(*-------------------------------------------------------------------------------------------------------ЕСЛИ ВТОРАЯ ГОРЕЛКА 1*)
	IF SECOND_GORELKA=1 THEN
		 IF AVARIA_OSNOVNAYA_GORELKA=FALSE  AND AVARIA_SECOND_GORELKA=FALSE THEN
			IF TEMPERATURA_2_OBR_OTOPLENIYA_AI_SP_307<TEMPERATURA_OFF_CIRCULACIONNOGO_NASOSA THEN
				xDO8:=TRUE;
				STEP_CIRCULAYCIONNUY_NASOS_1:=1;
			ELSE
				xDO8:=FALSE;
			END_IF
		END_IF
	END_IF
(*--------------------------------------------------------------------ЕСЛИ ВТОРАЯ ГОРЕЛКА 1 И ОСНОВНАЯ ВЫШЛА ИЗ СТРОЯ*)
	IF SECOND_GORELKA=1 THEN
		 IF AVARIA_OSNOVNAYA_GORELKA=TRUE  AND AVARIA_SECOND_GORELKA=FALSE THEN
			xDO8:=TRUE;
			STEP_CIRCULAYCIONNUY_NASOS_1:=1;
		END_IF
	END_IF
(*--------------------------------------------------------------------ЕСЛИ РЕЗЕРВНАЯ ГОРЕЛКА 1 И ВТОРАЯ ВЫШЛА ИЗ СТРОЯ*)
	IF RESERV_GORELKA=1 THEN
		 IF AVARIA_OSNOVNAYA_GORELKA=TRUE AND AVARIA_SECOND_GORELKA=TRUE THEN
			xDO8:=TRUE;
			STEP_CIRCULAYCIONNUY_NASOS_1:=1;
		END_IF
	END_IF
(*-------------------------------------------------------------------------------------------------------ЕСЛИ РЕЗЕРВНАЯ ГОРЕЛКА 1*)
	IF RESERV_GORELKA=1 THEN
		 IF TEMPERATURA_2_OBR_OTOPLENIYA_AI_SP_307<TEMPERATURA_OFF_CIRCULACIONNOGO_NASOSA THEN
				xDO8:=TRUE;
				STEP_CIRCULAYCIONNUY_NASOS_1:=1;
			ELSE
				xDO8:=FALSE;
			END_IF
	END_IF
END_IF
(*---------------------------------------------------------------------------------РАБОТА НАСОСОСА ПОСЛЕ ОСТАНОВКИ КОТЛА*)
IF PUSK_GORELKA_1=FALSE AND STEP_CIRCULAYCIONNUY_NASOS_1=1 THEN
	CASE STEP_CIRCULAYCIONNUY_NASOS_1 OF
		1:
			TIMER_CIRCUL_NASOS_1(IN:=TRUE,PT:=REAL_TO_TIME(VREMYA_RABOTU_CIRCULYACIONNOGO_NASOSA*1000));
				IF  TIMER_CIRCUL_NASOS_1.ET=TIMER_CIRCUL_NASOS_1.PT THEN
					STEP_CIRCULAYCIONNUY_NASOS_1:=0;
					TIMER_CIRCUL_NASOS_1(IN:=FALSE,PT:=T#0s);
      		 			TIMER_CIRCUL_NASOS_1;
					xDO8:=FALSE;
				END_IF
	END_CASE
ELSE
	TIMER_CIRCUL_NASOS_1(IN:=FALSE,PT:=T#0s);
      	TIMER_CIRCUL_NASOS_1;
END_IF
END_ACTION
ACTION CIRKULYACIONIY_NASOS_2:
IF PUSK_GORELKA_2=TRUE  THEN
(*---------------------------------------------------------------------------------------------------ЕСЛИ ОСНОВНАЯ ГОРЕЛКА 1*)
	IF  OSNOVNAYA_GORELKA=2  THEN
		xDO9:=TRUE;
		STEP_CIRCULAYCIONNUY_NASOS_2:=1;
	END_IF

(*-------------------------------------------------------------------------------------------------------ЕСЛИ ВТОРАЯ ГОРЕЛКА 1*)
	IF SECOND_GORELKA=2 THEN
		 IF AVARIA_OSNOVNAYA_GORELKA=FALSE  AND AVARIA_SECOND_GORELKA=FALSE THEN
			IF TEMPERATURA_2_OBR_OTOPLENIYA_AI_SP_307<TEMPERATURA_OFF_CIRCULACIONNOGO_NASOSA THEN
				xDO9:=TRUE;
				STEP_CIRCULAYCIONNUY_NASOS_2:=1;
			ELSE
				xDO9:=FALSE;
			END_IF
		END_IF
	END_IF
(*--------------------------------------------------------------------ЕСЛИ ВТОРАЯ ГОРЕЛКА 1 И ОСНОВНАЯ ВЫШЛА ИЗ СТРОЯ*)
	IF SECOND_GORELKA=2 THEN
		 IF AVARIA_OSNOVNAYA_GORELKA=TRUE  AND AVARIA_SECOND_GORELKA=FALSE THEN
			xDO9:=TRUE;
			STEP_CIRCULAYCIONNUY_NASOS_2:=1;
		END_IF
	END_IF
(*--------------------------------------------------------------------ЕСЛИ РЕЗЕРВНАЯ ГОРЕЛКА 1 И ВТОРАЯ ВЫШЛА ИЗ СТРОЯ*)
	IF RESERV_GORELKA=2 THEN
		 IF AVARIA_OSNOVNAYA_GORELKA=TRUE AND AVARIA_SECOND_GORELKA=TRUE THEN
			xDO9:=TRUE;
			STEP_CIRCULAYCIONNUY_NASOS_2:=1;
		END_IF
	END_IF
(*-------------------------------------------------------------------------------------------------------ЕСЛИ РЕЗЕРВНАЯ ГОРЕЛКА 1*)
	IF RESERV_GORELKA=2 THEN
		 IF TEMPERATURA_2_OBR_OTOPLENIYA_AI_SP_307<TEMPERATURA_OFF_CIRCULACIONNOGO_NASOSA THEN
				xDO9:=TRUE;
				STEP_CIRCULAYCIONNUY_NASOS_2:=1;
			ELSE
				xDO9:=FALSE;
			END_IF
	END_IF
END_IF
(*---------------------------------------------------------------------------------РАБОТА НАСОСОСА ПОСЛЕ ОСТАНОВКИ КОТЛА*)
IF PUSK_GORELKA_2=FALSE AND STEP_CIRCULAYCIONNUY_NASOS_2=1 THEN
	CASE STEP_CIRCULAYCIONNUY_NASOS_2 OF
		1:
			TIMER_CIRCUL_NASOS_2(IN:=TRUE,PT:=REAL_TO_TIME(VREMYA_RABOTU_CIRCULYACIONNOGO_NASOSA*1000));
				IF  TIMER_CIRCUL_NASOS_2.ET=TIMER_CIRCUL_NASOS_2.PT THEN
					STEP_CIRCULAYCIONNUY_NASOS_2:=0;
					TIMER_CIRCUL_NASOS_2(IN:=FALSE,PT:=T#0s);
      		 			TIMER_CIRCUL_NASOS_2;
					xDO9:=FALSE;
				END_IF
	END_CASE
ELSE
	TIMER_CIRCUL_NASOS_2(IN:=FALSE,PT:=T#0s);
      	TIMER_CIRCUL_NASOS_2;
END_IF
END_ACTION
ACTION CIRKULYACIONIY_NASOS_3:
IF PUSK_GORELKA_3=TRUE  THEN
(*---------------------------------------------------------------------------------------------------ЕСЛИ ОСНОВНАЯ ГОРЕЛКА 1*)
	IF  OSNOVNAYA_GORELKA=3  THEN
		xDO10:=TRUE;
		STEP_CIRCULAYCIONNUY_NASOS_3:=1;
	END_IF

(*-------------------------------------------------------------------------------------------------------ЕСЛИ ВТОРАЯ ГОРЕЛКА 1*)
	IF SECOND_GORELKA=3 THEN
		 IF AVARIA_OSNOVNAYA_GORELKA=FALSE  AND AVARIA_SECOND_GORELKA=FALSE THEN
			IF TEMPERATURA_2_OBR_OTOPLENIYA_AI_SP_307<TEMPERATURA_OFF_CIRCULACIONNOGO_NASOSA THEN
				xDO10:=TRUE;
				STEP_CIRCULAYCIONNUY_NASOS_3:=1;
			ELSE
				xDO10:=FALSE;
			END_IF
		END_IF
	END_IF
(*--------------------------------------------------------------------ЕСЛИ ВТОРАЯ ГОРЕЛКА 1 И ОСНОВНАЯ ВЫШЛА ИЗ СТРОЯ*)
	IF SECOND_GORELKA=3 THEN
		 IF AVARIA_OSNOVNAYA_GORELKA=TRUE  AND AVARIA_SECOND_GORELKA=FALSE THEN
			xDO10:=TRUE;
			STEP_CIRCULAYCIONNUY_NASOS_3:=1;
		END_IF
	END_IF
(*--------------------------------------------------------------------ЕСЛИ РЕЗЕРВНАЯ ГОРЕЛКА 1 И ВТОРАЯ ВЫШЛА ИЗ СТРОЯ*)
	IF RESERV_GORELKA=3 THEN
		 IF AVARIA_OSNOVNAYA_GORELKA=TRUE AND AVARIA_SECOND_GORELKA=TRUE THEN
			xDO10:=TRUE;
			STEP_CIRCULAYCIONNUY_NASOS_3:=1;
		END_IF
	END_IF
(*-------------------------------------------------------------------------------------------------------ЕСЛИ РЕЗЕРВНАЯ ГОРЕЛКА 1*)
	IF RESERV_GORELKA=3 THEN
		 IF TEMPERATURA_2_OBR_OTOPLENIYA_AI_SP_307<TEMPERATURA_OFF_CIRCULACIONNOGO_NASOSA THEN
				xDO10:=TRUE;
				STEP_CIRCULAYCIONNUY_NASOS_3:=1;
			ELSE
				xDO10:=FALSE;
			END_IF
	END_IF
END_IF
(*---------------------------------------------------------------------------------РАБОТА НАСОСОСА ПОСЛЕ ОСТАНОВКИ КОТЛА*)
IF PUSK_GORELKA_3=FALSE AND STEP_CIRCULAYCIONNUY_NASOS_3=1 THEN
	CASE STEP_CIRCULAYCIONNUY_NASOS_3 OF
		1:
			TIMER_CIRCUL_NASOS_3(IN:=TRUE,PT:=REAL_TO_TIME(VREMYA_RABOTU_CIRCULYACIONNOGO_NASOSA*1000));
				IF  TIMER_CIRCUL_NASOS_3.ET=TIMER_CIRCUL_NASOS_3.PT THEN
					STEP_CIRCULAYCIONNUY_NASOS_3:=0;
					TIMER_CIRCUL_NASOS_3(IN:=FALSE,PT:=T#0s);
      		 			TIMER_CIRCUL_NASOS_3;
					xDO10:=FALSE;
				END_IF
	END_CASE
ELSE
	TIMER_CIRCUL_NASOS_3(IN:=FALSE,PT:=T#0s);
      	TIMER_CIRCUL_NASOS_3;
END_IF
END_ACTION
ACTION DECOD_ERROR:
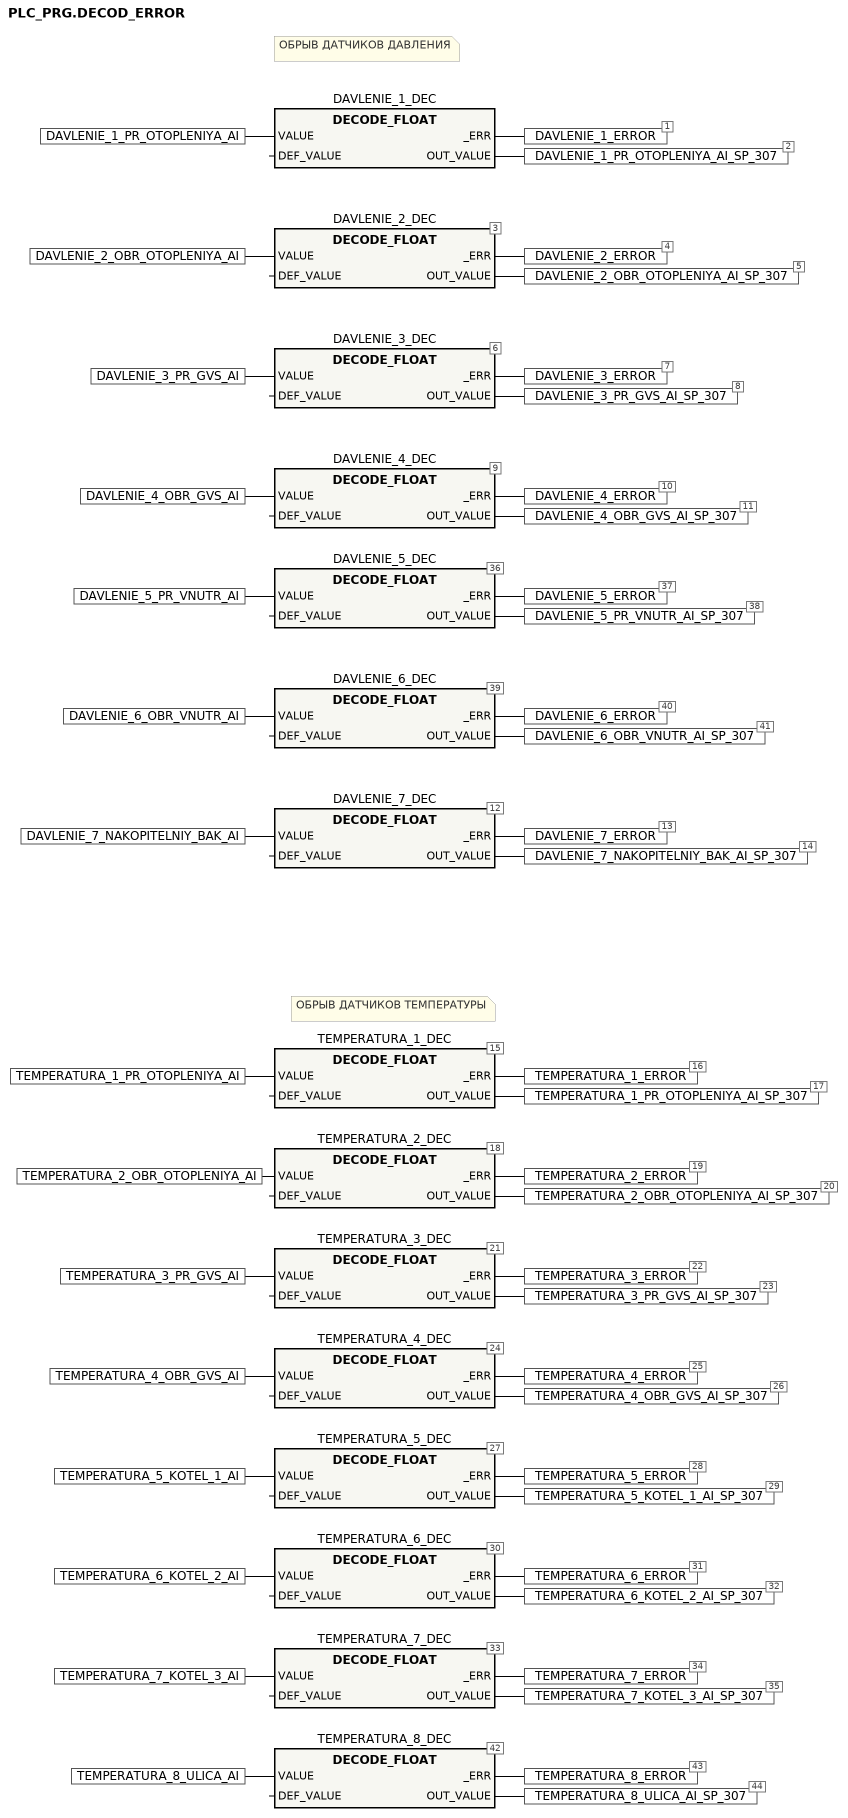
[picture p1: PLC_PRG.DECOD_ERROR (CFC)]
_CFC_ (* Continuous Function Chart, elements in execution order *)
(* ОБРЫВ ДАТЧИКОВ ДАВЛЕНИЯ *)
#0 DAVLENIE_1_DEC:DECODE_FLOAT(VALUE: DAVLENIE_1_PR_OTOPLENIYA_AI, DEF_VALUE: -)
#1 DAVLENIE_1_ERROR <= #0._ERR
#2 DAVLENIE_1_PR_OTOPLENIYA_AI_SP_307 <= #0.OUT_VALUE
#3 DAVLENIE_2_DEC:DECODE_FLOAT(VALUE: DAVLENIE_2_OBR_OTOPLENIYA_AI, DEF_VALUE: -)
#4 DAVLENIE_2_ERROR <= #3._ERR
#5 DAVLENIE_2_OBR_OTOPLENIYA_AI_SP_307 <= #3.OUT_VALUE
#6 DAVLENIE_3_DEC:DECODE_FLOAT(VALUE: DAVLENIE_3_PR_GVS_AI, DEF_VALUE: -)
#7 DAVLENIE_3_ERROR <= #6._ERR
#8 DAVLENIE_3_PR_GVS_AI_SP_307 <= #6.OUT_VALUE
#9 DAVLENIE_4_DEC:DECODE_FLOAT(VALUE: DAVLENIE_4_OBR_GVS_AI, DEF_VALUE: -)
#10 DAVLENIE_4_ERROR <= #9._ERR
#11 DAVLENIE_4_OBR_GVS_AI_SP_307 <= #9.OUT_VALUE
#12 DAVLENIE_7_DEC:DECODE_FLOAT(VALUE: DAVLENIE_7_NAKOPITELNIY_BAK_AI, DEF_VALUE: -)
#13 DAVLENIE_7_ERROR <= #12._ERR
#14 DAVLENIE_7_NAKOPITELNIY_BAK_AI_SP_307 <= #12.OUT_VALUE
#15 TEMPERATURA_1_DEC:DECODE_FLOAT(VALUE: TEMPERATURA_1_PR_OTOPLENIYA_AI, DEF_VALUE: -)
#16 TEMPERATURA_1_ERROR <= #15._ERR
#17 TEMPERATURA_1_PR_OTOPLENIYA_AI_SP_307 <= #15.OUT_VALUE
#18 TEMPERATURA_2_DEC:DECODE_FLOAT(VALUE: TEMPERATURA_2_OBR_OTOPLENIYA_AI, DEF_VALUE: -)
#19 TEMPERATURA_2_ERROR <= #18._ERR
#20 TEMPERATURA_2_OBR_OTOPLENIYA_AI_SP_307 <= #18.OUT_VALUE
#21 TEMPERATURA_3_DEC:DECODE_FLOAT(VALUE: TEMPERATURA_3_PR_GVS_AI, DEF_VALUE: -)
#22 TEMPERATURA_3_ERROR <= #21._ERR
#23 TEMPERATURA_3_PR_GVS_AI_SP_307 <= #21.OUT_VALUE
#24 TEMPERATURA_4_DEC:DECODE_FLOAT(VALUE: TEMPERATURA_4_OBR_GVS_AI, DEF_VALUE: -)
#25 TEMPERATURA_4_ERROR <= #24._ERR
#26 TEMPERATURA_4_OBR_GVS_AI_SP_307 <= #24.OUT_VALUE
#27 TEMPERATURA_5_DEC:DECODE_FLOAT(VALUE: TEMPERATURA_5_KOTEL_1_AI, DEF_VALUE: -)
#28 TEMPERATURA_5_ERROR <= #27._ERR
#29 TEMPERATURA_5_KOTEL_1_AI_SP_307 <= #27.OUT_VALUE
#30 TEMPERATURA_6_DEC:DECODE_FLOAT(VALUE: TEMPERATURA_6_KOTEL_2_AI, DEF_VALUE: -)
#31 TEMPERATURA_6_ERROR <= #30._ERR
#32 TEMPERATURA_6_KOTEL_2_AI_SP_307 <= #30.OUT_VALUE
#33 TEMPERATURA_7_DEC:DECODE_FLOAT(VALUE: TEMPERATURA_7_KOTEL_3_AI, DEF_VALUE: -)
#34 TEMPERATURA_7_ERROR <= #33._ERR
#35 TEMPERATURA_7_KOTEL_3_AI_SP_307 <= #33.OUT_VALUE
(* ОБРЫВ ДАТЧИКОВ ТЕМПЕРАТУРЫ *)
#36 DAVLENIE_5_DEC:DECODE_FLOAT(VALUE: DAVLENIE_5_PR_VNUTR_AI, DEF_VALUE: -)
#37 DAVLENIE_5_ERROR <= #36._ERR
#38 DAVLENIE_5_PR_VNUTR_AI_SP_307 <= #36.OUT_VALUE
#39 DAVLENIE_6_DEC:DECODE_FLOAT(VALUE: DAVLENIE_6_OBR_VNUTR_AI, DEF_VALUE: -)
#40 DAVLENIE_6_ERROR <= #39._ERR
#41 DAVLENIE_6_OBR_VNUTR_AI_SP_307 <= #39.OUT_VALUE
#42 TEMPERATURA_8_DEC:DECODE_FLOAT(VALUE: TEMPERATURA_8_ULICA_AI, DEF_VALUE: -)
#43 TEMPERATURA_8_ERROR <= #42._ERR
#44 TEMPERATURA_8_ULICA_AI_SP_307 <= #42.OUT_VALUE
_END_CFC_
(* the same logic as Structured Text *)
(* ОБРЫВ ДАТЧИКОВ ДАВЛЕНИЯ *)
DAVLENIE_1_DEC(VALUE := DAVLENIE_1_PR_OTOPLENIYA_AI);
DAVLENIE_1_ERROR := DAVLENIE_1_DEC._ERR;
DAVLENIE_1_PR_OTOPLENIYA_AI_SP_307 := DAVLENIE_1_DEC.OUT_VALUE;
DAVLENIE_2_DEC(VALUE := DAVLENIE_2_OBR_OTOPLENIYA_AI);
DAVLENIE_2_ERROR := DAVLENIE_2_DEC._ERR;
DAVLENIE_2_OBR_OTOPLENIYA_AI_SP_307 := DAVLENIE_2_DEC.OUT_VALUE;
DAVLENIE_3_DEC(VALUE := DAVLENIE_3_PR_GVS_AI);
DAVLENIE_3_ERROR := DAVLENIE_3_DEC._ERR;
DAVLENIE_3_PR_GVS_AI_SP_307 := DAVLENIE_3_DEC.OUT_VALUE;
DAVLENIE_4_DEC(VALUE := DAVLENIE_4_OBR_GVS_AI);
DAVLENIE_4_ERROR := DAVLENIE_4_DEC._ERR;
DAVLENIE_4_OBR_GVS_AI_SP_307 := DAVLENIE_4_DEC.OUT_VALUE;
DAVLENIE_7_DEC(VALUE := DAVLENIE_7_NAKOPITELNIY_BAK_AI);
DAVLENIE_7_ERROR := DAVLENIE_7_DEC._ERR;
DAVLENIE_7_NAKOPITELNIY_BAK_AI_SP_307 := DAVLENIE_7_DEC.OUT_VALUE;
TEMPERATURA_1_DEC(VALUE := TEMPERATURA_1_PR_OTOPLENIYA_AI);
TEMPERATURA_1_ERROR := TEMPERATURA_1_DEC._ERR;
TEMPERATURA_1_PR_OTOPLENIYA_AI_SP_307 := TEMPERATURA_1_DEC.OUT_VALUE;
TEMPERATURA_2_DEC(VALUE := TEMPERATURA_2_OBR_OTOPLENIYA_AI);
TEMPERATURA_2_ERROR := TEMPERATURA_2_DEC._ERR;
TEMPERATURA_2_OBR_OTOPLENIYA_AI_SP_307 := TEMPERATURA_2_DEC.OUT_VALUE;
TEMPERATURA_3_DEC(VALUE := TEMPERATURA_3_PR_GVS_AI);
TEMPERATURA_3_ERROR := TEMPERATURA_3_DEC._ERR;
TEMPERATURA_3_PR_GVS_AI_SP_307 := TEMPERATURA_3_DEC.OUT_VALUE;
TEMPERATURA_4_DEC(VALUE := TEMPERATURA_4_OBR_GVS_AI);
TEMPERATURA_4_ERROR := TEMPERATURA_4_DEC._ERR;
TEMPERATURA_4_OBR_GVS_AI_SP_307 := TEMPERATURA_4_DEC.OUT_VALUE;
TEMPERATURA_5_DEC(VALUE := TEMPERATURA_5_KOTEL_1_AI);
TEMPERATURA_5_ERROR := TEMPERATURA_5_DEC._ERR;
TEMPERATURA_5_KOTEL_1_AI_SP_307 := TEMPERATURA_5_DEC.OUT_VALUE;
TEMPERATURA_6_DEC(VALUE := TEMPERATURA_6_KOTEL_2_AI);
TEMPERATURA_6_ERROR := TEMPERATURA_6_DEC._ERR;
TEMPERATURA_6_KOTEL_2_AI_SP_307 := TEMPERATURA_6_DEC.OUT_VALUE;
TEMPERATURA_7_DEC(VALUE := TEMPERATURA_7_KOTEL_3_AI);
TEMPERATURA_7_ERROR := TEMPERATURA_7_DEC._ERR;
TEMPERATURA_7_KOTEL_3_AI_SP_307 := TEMPERATURA_7_DEC.OUT_VALUE;
(* ОБРЫВ ДАТЧИКОВ ТЕМПЕРАТУРЫ *)
DAVLENIE_5_DEC(VALUE := DAVLENIE_5_PR_VNUTR_AI);
DAVLENIE_5_ERROR := DAVLENIE_5_DEC._ERR;
DAVLENIE_5_PR_VNUTR_AI_SP_307 := DAVLENIE_5_DEC.OUT_VALUE;
DAVLENIE_6_DEC(VALUE := DAVLENIE_6_OBR_VNUTR_AI);
DAVLENIE_6_ERROR := DAVLENIE_6_DEC._ERR;
DAVLENIE_6_OBR_VNUTR_AI_SP_307 := DAVLENIE_6_DEC.OUT_VALUE;
TEMPERATURA_8_DEC(VALUE := TEMPERATURA_8_ULICA_AI);
TEMPERATURA_8_ERROR := TEMPERATURA_8_DEC._ERR;
TEMPERATURA_8_ULICA_AI_SP_307 := TEMPERATURA_8_DEC.OUT_VALUE;
END_ACTION
ACTION DO_DISKRETNUY_OUT:
xDO.0:=xDO0;
xDO.1:=xDO1;
xDO.2:=xDO2;
xDO.3:=xDO3;
xDO.4:=xDO4;
xDO.5:=xDO5;
xDO.6:=xDO6;
xDO.7:=xDO7;
xDO.8:=xDO8;
xDO.9:=xDO9;
xDO.10:=xDO10;
xDO.11:=xDO11;
xDO.12:=xDO12;
xDO.13:=xDO13;
xDO.14:=xDO14;
xDO.15:=xDO15;
END_ACTION
ACTION KASKAD_GORELOK:
UPRAVLENIE_GORELKOY_1;
UPRAVLENIE_GORELKOY_2;
UPRAVLENIE_GORELKOY_3;

IF WORK_KASKAD_1_SETEVOY=FALSE THEN
	PUSK_GORELKA_1:=FALSE;
	PUSK_GORELKA_2:=FALSE;
	PUSK_GORELKA_3:=FALSE;
END_IF
END_ACTION
ACTION MODUL_ERROR:
(*CASE STEP_MODUL_ERROR OF
0:
	IF ERROR_CONNECT<>0 THEN
		STEP_MODUL_ERROR:=1;
	END_IF
1:
	TIMER_MODUL_ERROR(IN:=TRUE, PT:=T#5s);
			IF  TIMER_MODUL_ERROR.ET=TIMER_MODUL_ERROR.PT THEN
				IF ERROR_CONNECT<>0 THEN
						ERROR_MODUL_SP_307:=TRUE;
						STEP_MODUL_ERROR:=0;
						TIMER_MODUL_ERROR(IN:=FALSE,PT:=T#0s);
      						TIMER_MODUL_ERROR;
				ELSE
					ERROR_MODUL_SP_307:=FALSE;
					STEP_MODUL_ERROR:=0;
					TIMER_MODUL_ERROR(IN:=FALSE,PT:=T#0s);
      					TIMER_MODUL_ERROR;
				END_IF
				TIMER_MODUL_ERROR(IN:=FALSE,PT:=T#0s);
      		 		TIMER_MODUL_ERROR;
			END_IF
END_CASE
*)

CASE STEP_MODUL_ERROR OF
0:
	IF ERROR_CONNECT<>0 THEN
		STEP_MODUL_ERROR:=1;
	END_IF
1:
	TIMER_MODUL_ERROR(IN:=TRUE, PT:=T#15s);
		IF  TIMER_MODUL_ERROR.ET=TIMER_MODUL_ERROR.PT THEN
			STEP_MODUL_ERROR:=2;
			TIMER_MODUL_ERROR(IN:=FALSE,PT:=T#0s);
      			TIMER_MODUL_ERROR;
		END_IF
	IF ERROR_CONNECT<>0 THEN
		KOLICHESTVO_OBRUV_MODUL:=KOLICHESTVO_OBRUV_MODUL+1;
	END_IF

2:
	IF KOLICHESTVO_OBRUV_MODUL>1000 THEN
		ERROR_MODUL_SP_307:=TRUE;
	ELSE
		ERROR_MODUL_SP_307:=FALSE;
		KOLICHESTVO_OBRUV_MODUL:=0;
		STEP_MODUL_ERROR:=0;
	END_IF
END_CASE
END_ACTION
ACTION NARABOTKA_MINUT:
NARABOTKA_CHASOV(PT:=T#60s, IN:= NOT NARABOTKA_CHASOV.Q); (*--------------------------------------ОБЩИЙ ТАЙМЕР*)

(*--------------------------------------------------------------------------------------------------КАСКАД НАСОСОСОВ. СЕТЕВОЙ*)

NARABOTKA_MINUT_KASKAD_1_NASOS_1_SETEVOY_SP_307:=NARABOTKA_MINUT_KASKAD_1_NASOS_1_SETEVOY_SP_307
									+ BOOL_TO_DWORD(NARABOTKA_CHASOV.Q AND WORK_KASKAD_1_SETEVOY AND xDO.0);

NARABOTKA_MINUT_KASKAD_1_NASOS_2_SETEVOY_SP_307:=NARABOTKA_MINUT_KASKAD_1_NASOS_2_SETEVOY_SP_307
 									+ BOOL_TO_DWORD(NARABOTKA_CHASOV.Q AND WORK_KASKAD_1_SETEVOY AND xDO.1);

(*---------------------------------------------------------------------------------------------------КАСКАД НАСОСОВ ВНУТРЕННИЙ*)
NARABOTKA_MINUT_KASKAD_2_VNUTR_NASOS_1_SP_307:=NARABOTKA_MINUT_KASKAD_2_VNUTR_NASOS_1_SP_307
									+ BOOL_TO_DWORD(NARABOTKA_CHASOV.Q AND WORK_KASKAD_2_VNUTR AND xDO.2);

NARABOTKA_MINUT_KASKAD_2_VNUTR_NASOS_2_SP_307:=NARABOTKA_MINUT_KASKAD_2_VNUTR_NASOS_2_SP_307
 									+ BOOL_TO_DWORD(NARABOTKA_CHASOV.Q AND WORK_KASKAD_2_VNUTR AND xDO.3);
(*--------------------------------------------------------------------------------------------------------КАСКАД НАСОСОСОВ. ГВС*)

NARABOTKA_MINUT_KASKAD_3_NASOS_1_GVS_SP_307:=NARABOTKA_MINUT_KASKAD_3_NASOS_1_GVS_SP_307
										 + BOOL_TO_DWORD(NARABOTKA_CHASOV.Q AND WORK_KASKAD_3_GVS AND xDO.4 );

NARABOTKA_MINUT_KASKAD_3_NASOS_2_GVS_SP_307:=NARABOTKA_MINUT_KASKAD_3_NASOS_2_GVS_SP_307
										+ BOOL_TO_DWORD(NARABOTKA_CHASOV.Q AND WORK_KASKAD_3_GVS AND xDO.5 );

(*------------------------------------------------------------------------------------------------КАСКАД НАСОСОСОВ. ПОДПИТКА*)

NARABOTKA_MINUT_KASKAD_4_NASOS_1_PODPITKA_SP_307:=NARABOTKA_MINUT_KASKAD_4_NASOS_1_PODPITKA_SP_307
									 + BOOL_TO_DWORD(NARABOTKA_CHASOV.Q AND WORK_KASKAD_4_PODPITKA AND xDO.6 );

NARABOTKA_MINUT_KASKAD_4_NASOS_2_PODPITKA_SP_307:=NARABOTKA_MINUT_KASKAD_4_NASOS_2_PODPITKA_SP_307
									+ BOOL_TO_DWORD(NARABOTKA_CHASOV.Q AND WORK_KASKAD_4_PODPITKA AND xDO.7 );

(*------------------------------------------------------------------------------------------------------ЦИРКУЛЯЦИОННЫЕ НАСОСЫ*)

NARABOTKA_MINUT_KASKAD_5_NASOS_1_CIRKUL_SP_307:=NARABOTKA_MINUT_KASKAD_5_NASOS_1_CIRKUL_SP_307
									 + BOOL_TO_DWORD(NARABOTKA_CHASOV.Q AND xDO.8 );

NARABOTKA_MINUT_KASKAD_5_NASOS_2_CIRKUL_SP_307:=NARABOTKA_MINUT_KASKAD_5_NASOS_2_CIRKUL_SP_307
									 + BOOL_TO_DWORD(NARABOTKA_CHASOV.Q AND xDO.9 );

NARABOTKA_MINUT_KASKAD_5_NASOS_3_CIRKUL_SP_307:=NARABOTKA_MINUT_KASKAD_5_NASOS_3_CIRKUL_SP_307
									 + BOOL_TO_DWORD(NARABOTKA_CHASOV.Q AND xDO.10 );
(*--------------------------------------------------------------------------------------------------------------------------ГОРЕЛКА 1*)

NARABOTKA_MINUT_GORELKA_1_SP_307:=NARABOTKA_MINUT_GORELKA_1_SP_307
															+BOOL_TO_DWORD(NARABOTKA_CHASOV.Q AND WORK_GORELKA_1);

(*--------------------------------------------------------------------------------------------------------------------------ГОРЕЛКА 2*)

NARABOTKA_MINUT_GORELKA_2_SP_307:=NARABOTKA_MINUT_GORELKA_2_SP_307
															+BOOL_TO_DWORD(NARABOTKA_CHASOV.Q AND WORK_GORELKA_2);

(*--------------------------------------------------------------------------------------------------------------------------ГОРЕЛКА 3*)

NARABOTKA_MINUT_GORELKA_3_SP_307:=NARABOTKA_MINUT_GORELKA_3_SP_307
															+BOOL_TO_DWORD(NARABOTKA_CHASOV.Q AND WORK_GORELKA_3);
END_ACTION
ACTION NARABOTKA_VKLUCHENIY:
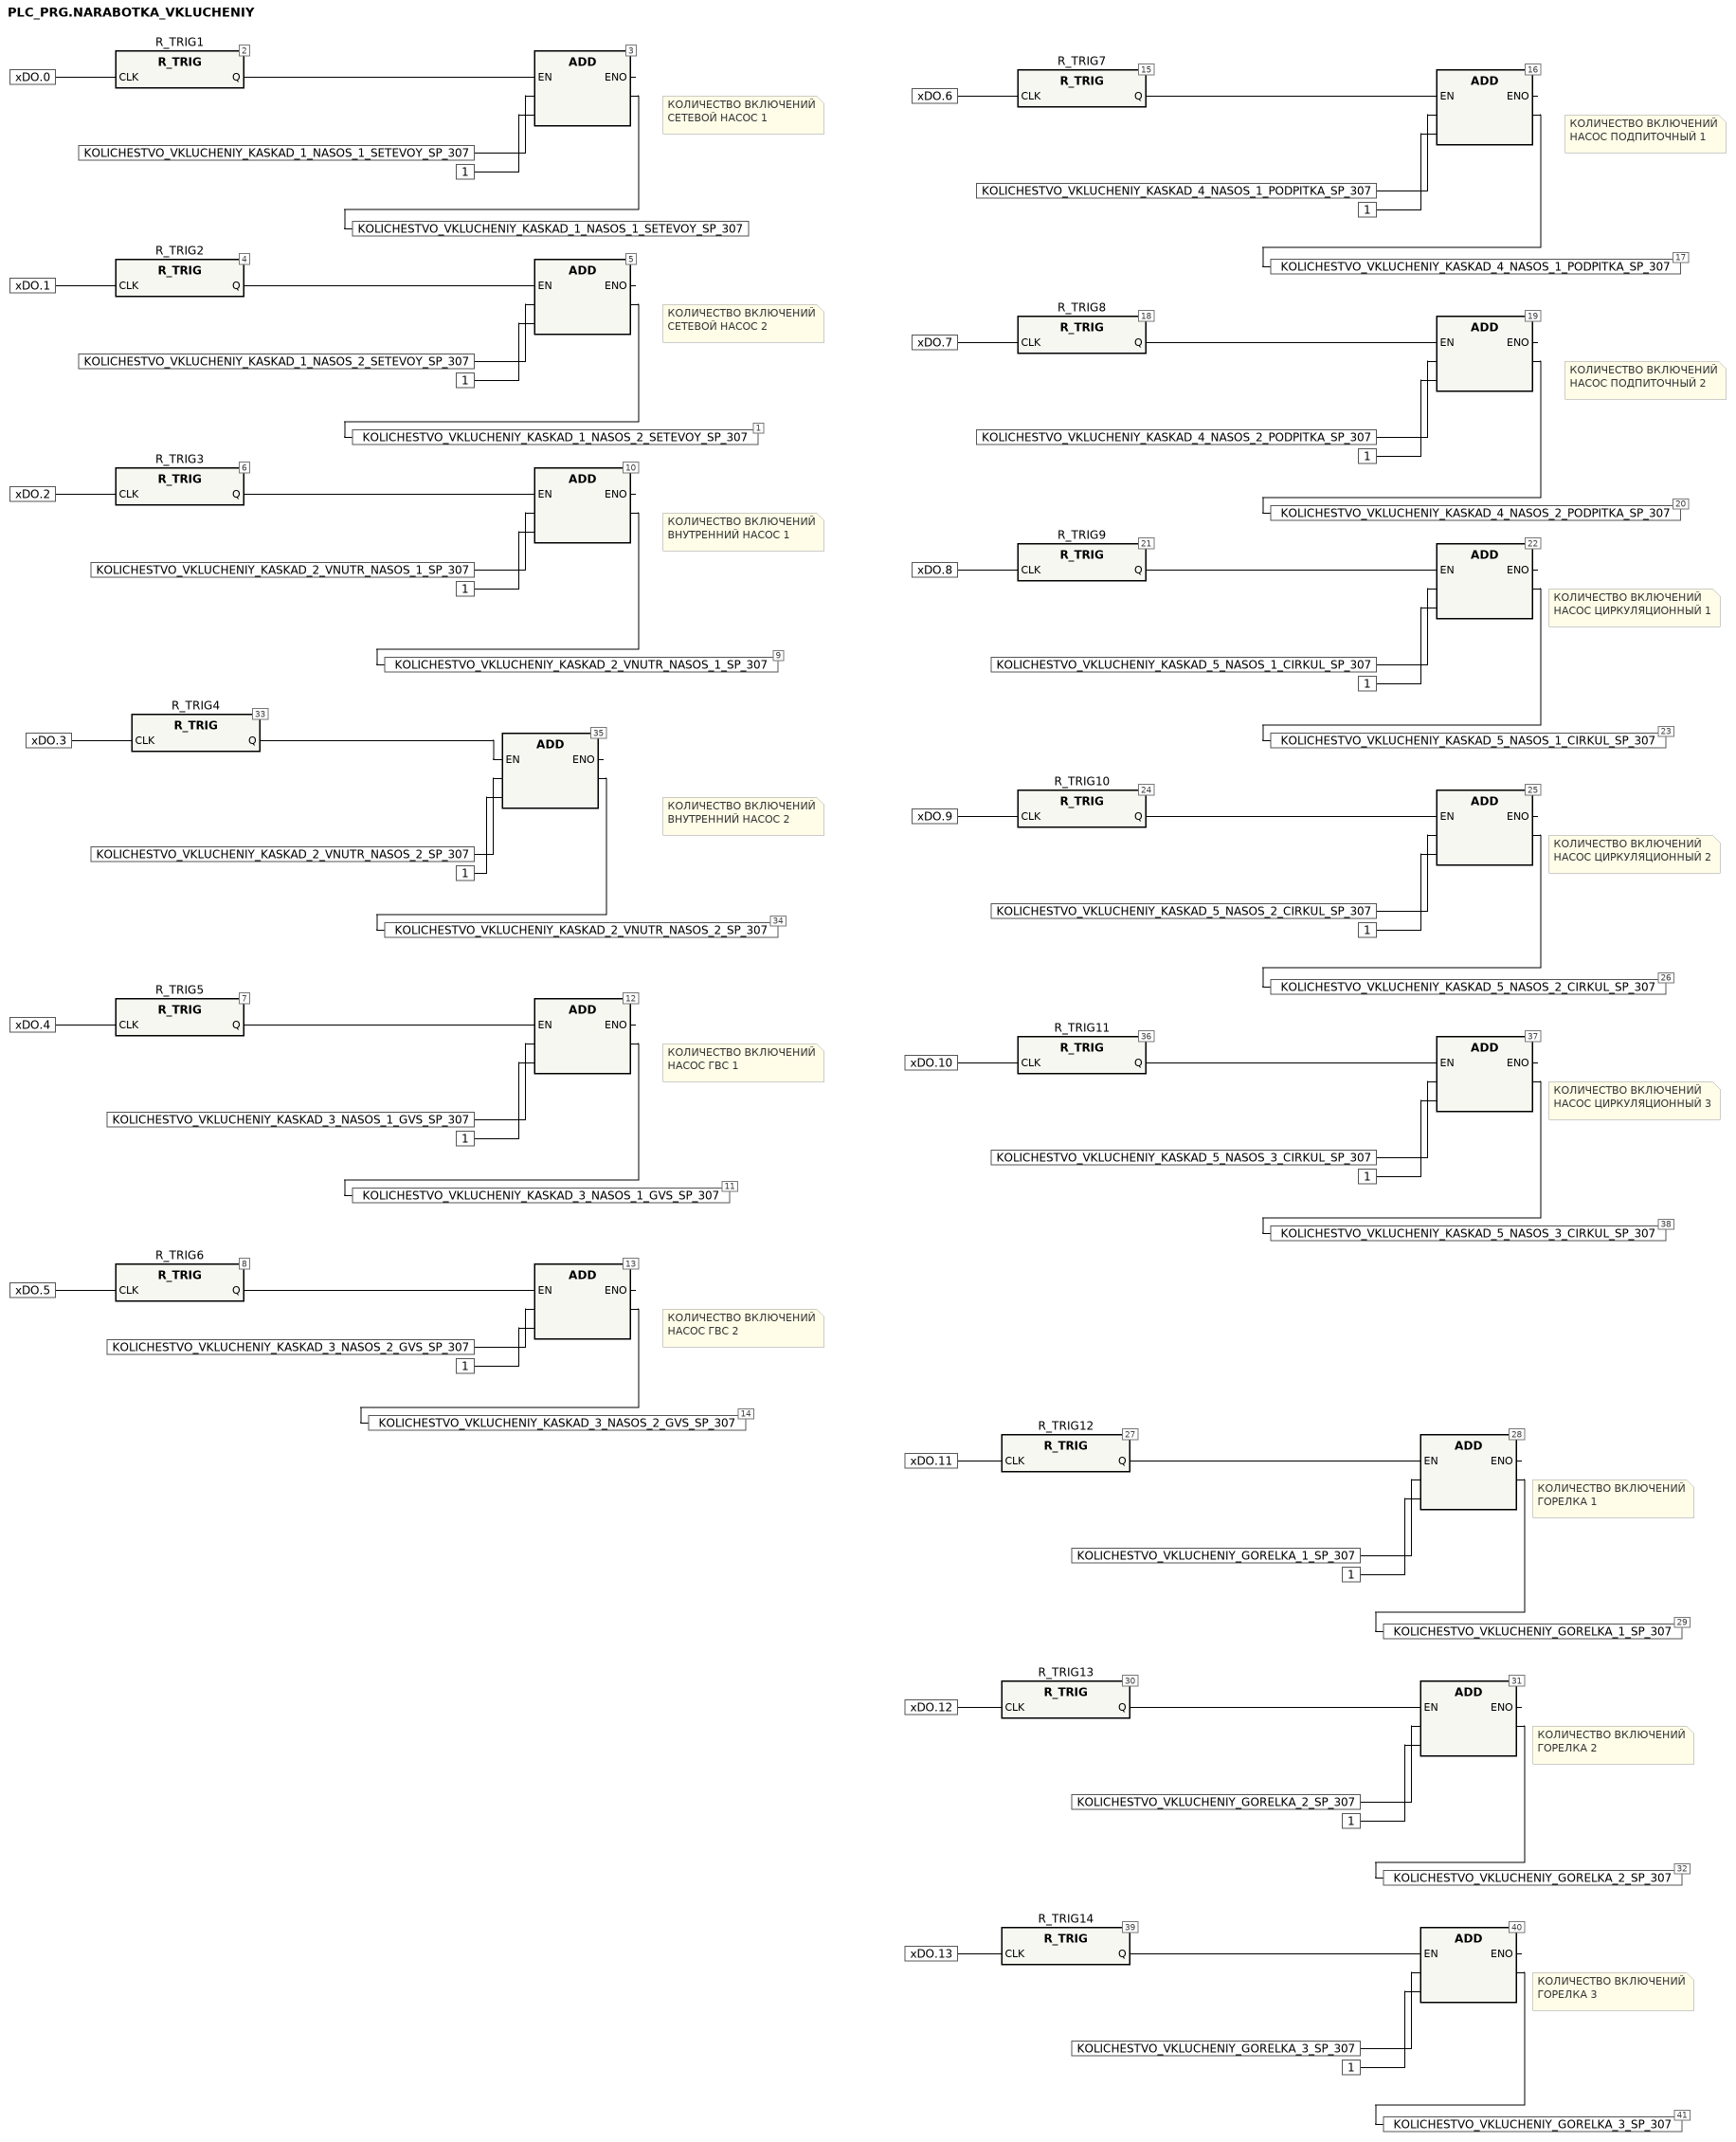
_CFC_ (* Continuous Function Chart, elements in execution order *)
(* КОЛИЧЕСТВО ВКЛЮЧЕНИЙ / СЕТЕВОЙ НАСОС 1 *)
#0 KOLICHESTVO_VKLUCHENIY_KASKAD_1_NASOS_1_SETEVOY_SP_307 <= #3
#1 KOLICHESTVO_VKLUCHENIY_KASKAD_1_NASOS_2_SETEVOY_SP_307 <= #5
#2 R_TRIG1:R_TRIG(CLK: xDO.0)
#3 ADD(EN: #2.Q, KOLICHESTVO_VKLUCHENIY_KASKAD_1_NASOS_1_SETEVOY_SP_307, 1)
#4 R_TRIG2:R_TRIG(CLK: xDO.1)
#5 ADD(EN: #4.Q, KOLICHESTVO_VKLUCHENIY_KASKAD_1_NASOS_2_SETEVOY_SP_307, 1)
#6 R_TRIG3:R_TRIG(CLK: xDO.2)
#7 R_TRIG5:R_TRIG(CLK: xDO.4)
#8 R_TRIG6:R_TRIG(CLK: xDO.5)
(* КОЛИЧЕСТВО ВКЛЮЧЕНИЙ / СЕТЕВОЙ НАСОС 2 *)
#9 KOLICHESTVO_VKLUCHENIY_KASKAD_2_VNUTR_NASOS_1_SP_307 <= #10
#10 ADD(EN: #6.Q, KOLICHESTVO_VKLUCHENIY_KASKAD_2_VNUTR_NASOS_1_SP_307, 1)
(* КОЛИЧЕСТВО ВКЛЮЧЕНИЙ / ВНУТРЕННИЙ НАСОС 1 *)
#11 KOLICHESTVO_VKLUCHENIY_KASKAD_3_NASOS_1_GVS_SP_307 <= #12
#12 ADD(EN: #7.Q, KOLICHESTVO_VKLUCHENIY_KASKAD_3_NASOS_1_GVS_SP_307, 1)
(* КОЛИЧЕСТВО ВКЛЮЧЕНИЙ / НАСОС ГВС 1 *)
#13 ADD(EN: #8.Q, KOLICHESTVO_VKLUCHENIY_KASKAD_3_NASOS_2_GVS_SP_307, 1)
(* КОЛИЧЕСТВО ВКЛЮЧЕНИЙ / НАСОС ГВС 2 *)
#14 KOLICHESTVO_VKLUCHENIY_KASKAD_3_NASOS_2_GVS_SP_307 <= #13
#15 R_TRIG7:R_TRIG(CLK: xDO.6)
#16 ADD(EN: #15.Q, KOLICHESTVO_VKLUCHENIY_KASKAD_4_NASOS_1_PODPITKA_SP_307, 1)
(* КОЛИЧЕСТВО ВКЛЮЧЕНИЙ / НАСОС ПОДПИТОЧНЫЙ 1 *)
#17 KOLICHESTVO_VKLUCHENIY_KASKAD_4_NASOS_1_PODPITKA_SP_307 <= #16
#18 R_TRIG8:R_TRIG(CLK: xDO.7)
#19 ADD(EN: #18.Q, KOLICHESTVO_VKLUCHENIY_KASKAD_4_NASOS_2_PODPITKA_SP_307, 1)
(* КОЛИЧЕСТВО ВКЛЮЧЕНИЙ / НАСОС ПОДПИТОЧНЫЙ 2 *)
#20 KOLICHESTVO_VKLUCHENIY_KASKAD_4_NASOS_2_PODPITKA_SP_307 <= #19
#21 R_TRIG9:R_TRIG(CLK: xDO.8)
#22 ADD(EN: #21.Q, KOLICHESTVO_VKLUCHENIY_KASKAD_5_NASOS_1_CIRKUL_SP_307, 1)
(* КОЛИЧЕСТВО ВКЛЮЧЕНИЙ / НАСОС ЦИРКУЛЯЦИОННЫЙ 1 *)
#23 KOLICHESTVO_VKLUCHENIY_KASKAD_5_NASOS_1_CIRKUL_SP_307 <= #22
#24 R_TRIG10:R_TRIG(CLK: xDO.9)
#25 ADD(EN: #24.Q, KOLICHESTVO_VKLUCHENIY_KASKAD_5_NASOS_2_CIRKUL_SP_307, 1)
(* КОЛИЧЕСТВО ВКЛЮЧЕНИЙ / НАСОС ЦИРКУЛЯЦИОННЫЙ 2 *)
#26 KOLICHESTVO_VKLUCHENIY_KASKAD_5_NASOS_2_CIRKUL_SP_307 <= #25
#27 R_TRIG12:R_TRIG(CLK: xDO.11)
#28 ADD(EN: #27.Q, KOLICHESTVO_VKLUCHENIY_GORELKA_1_SP_307, 1)
(* КОЛИЧЕСТВО ВКЛЮЧЕНИЙ / ГОРЕЛКА 1 *)
#29 KOLICHESTVO_VKLUCHENIY_GORELKA_1_SP_307 <= #28
#30 R_TRIG13:R_TRIG(CLK: xDO.12)
#31 ADD(EN: #30.Q, KOLICHESTVO_VKLUCHENIY_GORELKA_2_SP_307, 1)
(* КОЛИЧЕСТВО ВКЛЮЧЕНИЙ / ГОРЕЛКА 2 *)
#32 KOLICHESTVO_VKLUCHENIY_GORELKA_2_SP_307 <= #31
#33 R_TRIG4:R_TRIG(CLK: xDO.3)
#34 KOLICHESTVO_VKLUCHENIY_KASKAD_2_VNUTR_NASOS_2_SP_307 <= #35
#35 ADD(EN: #33.Q, KOLICHESTVO_VKLUCHENIY_KASKAD_2_VNUTR_NASOS_2_SP_307, 1)
(* КОЛИЧЕСТВО ВКЛЮЧЕНИЙ / ВНУТРЕННИЙ НАСОС 2 *)
#36 R_TRIG11:R_TRIG(CLK: xDO.10)
#37 ADD(EN: #36.Q, KOLICHESTVO_VKLUCHENIY_KASKAD_5_NASOS_3_CIRKUL_SP_307, 1)
(* КОЛИЧЕСТВО ВКЛЮЧЕНИЙ / НАСОС ЦИРКУЛЯЦИОННЫЙ 3 *)
#38 KOLICHESTVO_VKLUCHENIY_KASKAD_5_NASOS_3_CIRKUL_SP_307 <= #37
#39 R_TRIG14:R_TRIG(CLK: xDO.13)
#40 ADD(EN: #39.Q, KOLICHESTVO_VKLUCHENIY_GORELKA_3_SP_307, 1)
(* КОЛИЧЕСТВО ВКЛЮЧЕНИЙ / ГОРЕЛКА 3 *)
#41 KOLICHESTVO_VKLUCHENIY_GORELKA_3_SP_307 <= #40
_END_CFC_
END_ACTION
ACTION OBRABOTKA_AVARIY:
(*
	xDO0,(*---------------------------------------------------------------------------------------------------------НАСОС СЕТЕВОЙ 1*)
	xDO1,(*---------------------------------------------------------------------------------------------------------НАСОС СЕТЕВОЙ 2*)
	xDO2,(*----------------------------------------------------------------------------------------НАСОС ВНУТРЕННЕГО КОНТУРА 1*)
	xDO3,(*----------------------------------------------------------------------------------------НАСОС ВНУТРЕННЕГО КОНТУРА 2*)
	xDO4,(*---------------------------------------------------------------------------------------------------------------НАСОС ГВС 1*)
	xDO5,(*---------------------------------------------------------------------------------------------------------------НАСОС ГВС 2*)
	xDO6,(*--------------------------------------------------------------------------------------------------НАСОС ПОДПИТОЧНЫЙ 1*)
	xDO7,(*--------------------------------------------------------------------------------------------------НАСОС ПОДПИТОЧНЫЙ 2*)
	xDO8,(*----------------------------------------------------------------------------------------------НАСОС ЦИРКУЛЯЦИОННЫЙ 1*)
	xDO9, (*---------------------------------------------------------------------------------------------НАСОС ЦИРКУЛЯЦИОННЫЙ 2*)
	xDO10,(*--------------------------------------------------------------------------------------------НАСОС ЦИРКУЛЯЦИОННЫЙ 3*)
	xDO11,(*-------------------------------------------------------------------------------------------------ГОРЕЛКА 1: ТЕРМОСТАТ*)
	xDO12,(*-------------------------------------------------------------------------------------------------ГОРЕЛКА 2: ТЕРМОСТАТ*)
	xDO13,(*-------------------------------------------------------------------------------------------------ГОРЕЛКА 3: ТЕРМОСТАТ*)
	xDO14,(*------------------------------------------------------------*)
	xDO15:(*------------------------------------------------------------*)
*)



(*--------------------------------------------------------------------------------------ЕСЛИ АВАРИЯ ОБРЫВА ФАЗ ИЛИ ПЕРЕКОС ФАЗ*)
IF AVARIA_PHASA_SP_307 OR AVARIA_FIRE_SP_307 OR AVARIA_GAZ_SP_307 THEN
	xDO.0:=xDO0:=FALSE;(*---------------------------------------------------------------------------------------НАСОС СЕТЕВОЙ 1*)
	xDO.1:=xDO1:=FALSE;(*---------------------------------------------------------------------------------------НАСОС СЕТЕВОЙ 2*)
	xDO.2:=xDO2:=FALSE;(*----------------------------------------------------------------------НАСОС ВНУТРЕННЕГО КОНТУРА 1*)
	xDO.3:=xDO3:=FALSE;(*----------------------------------------------------------------------НАСОС ВНУТРЕННЕГО КОНТУРА 2*)
	xDO.4:=xDO4:=FALSE;(*---------------------------------------------------------------------------------------------НАСОС ГВС 1*)
	xDO.5:=xDO5:=FALSE;(*---------------------------------------------------------------------------------------------НАСОС ГВС 2*)
	xDO.6:=xDO6:=FALSE;(*--------------------------------------------------------------------------------НАСОС ПОДПИТОЧНЫЙ 1*)
	xDO.7:=xDO7:=FALSE;(*--------------------------------------------------------------------------------НАСОС ПОДПИТОЧНЫЙ 2*)
	(*
	xDO.8:=xDO8:=FALSE;(*----------------------------------------------------------------------------НАСОС ЦИРКУЛЯЦИОННЫЙ 1*)
	xDO.9:=xDO9:=FALSE;(*----------------------------------------------------------------------------НАСОС ЦИРКУЛЯЦИОННЫЙ 2*)
	xDO.10:=xDO10:=FALSE;(*-------------------------------------------------------------------------НАСОС ЦИРКУЛЯЦИОННЫЙ 3*)
	*)
	xDO.11:=xDO11:=FALSE;(*------------------------------------------------------------------------------ГОРЕЛКА 1: ТЕРМОСТАТ*)
	xDO.12:=xDO12:=FALSE;(*------------------------------------------------------------------------------ГОРЕЛКА 2: ТЕРМОСТАТ*)
	xDO.13:=xDO13:=FALSE;(*------------------------------------------------------------------------------ГОРЕЛКА 3: ТЕРМОСТАТ*)
	xDO.14:=xDO14:=FALSE;
	xDO.15:=xDO15:=FALSE;

	PUSK_GORELKA_1:=FALSE;
	PUSK_GORELKA_2:=FALSE;
	PUSK_GORELKA_3:=FALSE;
	PUSK_KASKAD_NASOSOV_1_SETEVOY:=FALSE;
	PUSK_KASKAD_NASOSOV_2_VNUTR:=FALSE;
	PUSK_KASKAD_NASOSOV_3_GVS:=FALSE;
	PUSK_KASKAD_NASOSOV_4_PODPITKA:=FALSE;

	STEP_MAIN:=0;
	STEP_DAVL_POKOYA:=0;
	STEP3:=0;
	STEP4:=0;
	STEP_SBROS_GVS:=0;
	STEP_SBROS_OTOPLENIYA:=0;
	STEP_PODOGREV_SECOND_GORELKA:=0;
	STEP_PODOGREV_RESERV_GORELKA:=0;
	STEP_AVARIA_PODOGREV_RESERV_GORELKA:=0;
END_IF
(*-----------------------------------------------------------------------------------------------------------------ЕСЛИ АВАРИЯ ПОЖАР*)
(*
IF AVARIA_FIRE_SP_307 THEN
	xDO.0:=xDO0:=FALSE;(*---------------------------------------------------------------------------------------НАСОС СЕТЕВОЙ 1*)
	xDO.1:=xDO1:=FALSE;(*---------------------------------------------------------------------------------------НАСОС СЕТЕВОЙ 2*)
	xDO.2:=xDO2:=FALSE;(*-------------------------------------------------------------------------------------------НАСОС ЛЕТНИЙ*)
	xDO.3:=xDO3:=FALSE;(*----------------------------------------------------------------------------------------------НАСОС ГВС 1*)
	xDO.4:=xDO4:=FALSE;(*----------------------------------------------------------------------------------------------НАСОС ГВС 2*)
	xDO.5:=xDO5:=FALSE;(*--------------------------------------------------------------------------------НАСОС ПОДПИТОЧНЫЙ 1*)
	xDO.6:=xDO6:=FALSE;(*--------------------------------------------------------------------------------НАСОС ПОДПИТОЧНЫЙ 2*)
	(*xDO.7:=xDO7:=FALSE;(*-----------------------------------------------------------------------НАСОС ЦИРКУЛЯЦИОННЫЙ 1*)*)
	(*xDO.8:=xDO8:=FALSE;(*-----------------------------------------------------------------------НАСОС ЦИРКУЛЯЦИОННЫЙ 2*)*)
	xDO.9:=xDO9:=FALSE;(*-------------------------------------------------------------КЛАПАН ЭЛЕКТРОМАГНИТНЫЙ ПОДПИТКИ*)
	xDO.10:=xDO10:=FALSE;(*---------------------------------------------КЛАПАН ЭЛЕКТРОМАГНИТНЫЙ НАКОПИТЕЛЬНЫЙ БАК*)
	xDO.11:=xDO11:=FALSE;(*----------------------------------------------------КЛАПАН ЭЛЕКТРОМАГНИТНЫЙ ОТСЕЧНОЙ ГАЗА*)
	xDO.12:=xDO12:=FALSE;(*---------------------------------------------------------------------------------------ПУСК ГОРЕЛКИ 1*)
	xDO.13:=xDO13:=FALSE;(*---------------------------------------------------------------------------------------ПУСК ГОРЕЛКИ 2*)
	xDO.14:=xDO14:=FALSE;(*-------------------------------------------------------------------------БОЛЬШОЕ ПЛАМЯ ГОРЕЛКИ 1*)
	xDO.15:=xDO15:=FALSE;(*-------------------------------------------------------------------------БОЛЬШОЕ ПЛАМЯ ГОРЕЛКИ 2*)

	PUSK_GORELKA_1:=FALSE;
	PUSK_GORELKA_2:=FALSE;
	PUSK_KASKAD_NASOSOV_1_SETEVOY:=FALSE;
	(*PUSK_KASKAD_NASOSOV_2_LETNIY:=FALSE;-----------------------------------------------------------------------------------------------------------УДАЛИТЬ*)
	PUSK_KASKAD_NASOSOV_3_GVS:=FALSE;
	PUSK_KASKAD_NASOSOV_4_PODPITKA:=FALSE;
END_IF
*)
(*---------------------------------------------------------------------------------------------------------------------ЕСЛИ АВАРИЯ ГАЗ*)
(*
IF AVARIA_GAZ_SP_307 THEN
	xDO.0:=xDO0:=FALSE;(*---------------------------------------------------------------------------------------НАСОС СЕТЕВОЙ 1*)
	xDO.1:=xDO1:=FALSE;(*---------------------------------------------------------------------------------------НАСОС СЕТЕВОЙ 2*)
	xDO.2:=xDO2:=FALSE;(*-------------------------------------------------------------------------------------------НАСОС ЛЕТНИЙ*)
	xDO.3:=xDO3:=FALSE;(*----------------------------------------------------------------------------------------------НАСОС ГВС 1*)
	xDO.4:=xDO4:=FALSE;(*----------------------------------------------------------------------------------------------НАСОС ГВС 2*)
	xDO.5:=xDO5:=FALSE;(*--------------------------------------------------------------------------------НАСОС ПОДПИТОЧНЫЙ 1*)
	xDO.6:=xDO6:=FALSE;(*--------------------------------------------------------------------------------НАСОС ПОДПИТОЧНЫЙ 2*)
	(*xDO.7:=xDO7:=FALSE;(*-----------------------------------------------------------------------НАСОС ЦИРКУЛЯЦИОННЫЙ 1*)*)
	(*xDO.8:=xDO8:=FALSE;(*-----------------------------------------------------------------------НАСОС ЦИРКУЛЯЦИОННЫЙ 2*)*)
	xDO.9:=xDO9:=FALSE;(*-------------------------------------------------------------КЛАПАН ЭЛЕКТРОМАГНИТНЫЙ ПОДПИТКИ*)
	xDO.10:=xDO10:=FALSE;(*---------------------------------------------КЛАПАН ЭЛЕКТРОМАГНИТНЫЙ НАКОПИТЕЛЬНЫЙ БАК*)
	xDO.11:=xDO11:=FALSE;(*----------------------------------------------------КЛАПАН ЭЛЕКТРОМАГНИТНЫЙ ОТСЕЧНОЙ ГАЗА*)
	xDO.12:=xDO12:=FALSE;(*---------------------------------------------------------------------------------------ПУСК ГОРЕЛКИ 1*)
	xDO.13:=xDO13:=FALSE;(*---------------------------------------------------------------------------------------ПУСК ГОРЕЛКИ 2*)
	xDO.14:=xDO14:=FALSE;(*-------------------------------------------------------------------------БОЛЬШОЕ ПЛАМЯ ГОРЕЛКИ 1*)
	xDO.15:=xDO15:=FALSE;(*-------------------------------------------------------------------------БОЛЬШОЕ ПЛАМЯ ГОРЕЛКИ 2*)

	PUSK_GORELKA_1:=FALSE;
	PUSK_GORELKA_2:=FALSE;
	PUSK_KASKAD_NASOSOV_1_SETEVOY:=FALSE;
	(*PUSK_KASKAD_NASOSOV_2_LETNIY:=FALSE;-----------------------------------------------------------------------------------------------------------УДАЛИТЬ*)
	PUSK_KASKAD_NASOSOV_3_GVS:=FALSE;
	PUSK_KASKAD_NASOSOV_4_PODPITKA:=FALSE;
END_IF
*)

(*--------------------------------------------------------------------------------ЕСЛИ АВАРИЯ ВЫСОКАЯ ТЕМПЕРАТУРА ГОРЕЛКИ 1*)
IF AVARIA_VUSOKAYA_TEMPERATURA_KOTEL_1_SP_307 THEN

	xDO.11:=xDO11:=FALSE;(*------------------------------------------------------------------------------ГОРЕЛКА 1: ТЕРМОСТАТ*)
	xDO.12:=xDO12:=FALSE;(*------------------------------------------------------------------------------ГОРЕЛКА 2: ТЕРМОСТАТ*)
	xDO.13:=xDO13:=FALSE;(*------------------------------------------------------------------------------ГОРЕЛКА 3: ТЕРМОСТАТ*)
	xDO.14:=xDO14:=FALSE;
	xDO.15:=xDO15:=FALSE;

	PUSK_GORELKA_1:=FALSE;
	PUSK_GORELKA_2:=FALSE;
	PUSK_GORELKA_3:=FALSE;

END_IF
(*--------------------------------------------------------------------------------ЕСЛИ АВАРИЯ ВЫСОКАЯ ТЕМПЕРАТУРА ГОРЕЛКИ 2*)
IF AVARIA_VUSOKAYA_TEMPERATURA_KOTEL_2_SP_307 THEN
	xDO.11:=xDO11:=FALSE;(*------------------------------------------------------------------------------ГОРЕЛКА 1: ТЕРМОСТАТ*)
	xDO.12:=xDO12:=FALSE;(*------------------------------------------------------------------------------ГОРЕЛКА 2: ТЕРМОСТАТ*)
	xDO.13:=xDO13:=FALSE;(*------------------------------------------------------------------------------ГОРЕЛКА 3: ТЕРМОСТАТ*)
	xDO.14:=xDO14:=FALSE;
	xDO.15:=xDO15:=FALSE;

	PUSK_GORELKA_1:=FALSE;
	PUSK_GORELKA_2:=FALSE;
	PUSK_GORELKA_3:=FALSE;
END_IF
(*--------------------------------------------------------------------------------ЕСЛИ АВАРИЯ ВЫСОКАЯ ТЕМПЕРАТУРА ГОРЕЛКИ 2*)
IF AVARIA_VUSOKAYA_TEMPERATURA_KOTEL_3_SP_307 THEN
	xDO.11:=xDO11:=FALSE;(*------------------------------------------------------------------------------ГОРЕЛКА 1: ТЕРМОСТАТ*)
	xDO.12:=xDO12:=FALSE;(*------------------------------------------------------------------------------ГОРЕЛКА 2: ТЕРМОСТАТ*)
	xDO.13:=xDO13:=FALSE;(*------------------------------------------------------------------------------ГОРЕЛКА 3: ТЕРМОСТАТ*)
	xDO.14:=xDO14:=FALSE;
	xDO.15:=xDO15:=FALSE;

	PUSK_GORELKA_1:=FALSE;
	PUSK_GORELKA_2:=FALSE;
	PUSK_GORELKA_3:=FALSE;
END_IF

(*----------------------------------------------------------------------------------ЕСЛИ АВАРИЯ ВЫСОКОЕ ДАВЛЕНИЕ ОТОПЛЕНИЯ*)
IF AVARIA_VUSOKOE_DAVLENIE_OTOPLENIYA_SP_307 THEN
	xDO.0:=xDO0:=FALSE;(*---------------------------------------------------------------------------------------НАСОС СЕТЕВОЙ 1*)
	xDO.1:=xDO1:=FALSE;(*---------------------------------------------------------------------------------------НАСОС СЕТЕВОЙ 2*)
	(*
	xDO.2:=xDO2:=FALSE;(*----------------------------------------------------------------------НАСОС ВНУТРЕННЕГО КОНТУРА 1*)
	xDO.3:=xDO3:=FALSE;(*----------------------------------------------------------------------НАСОС ВНУТРЕННЕГО КОНТУРА 2*)
	*)
	xDO.11:=xDO11:=FALSE;(*------------------------------------------------------------------------------ГОРЕЛКА 1: ТЕРМОСТАТ*)
	xDO.12:=xDO12:=FALSE;(*------------------------------------------------------------------------------ГОРЕЛКА 2: ТЕРМОСТАТ*)
	xDO.13:=xDO13:=FALSE;(*------------------------------------------------------------------------------ГОРЕЛКА 3: ТЕРМОСТАТ*)


	PUSK_GORELKA_1:=FALSE;
	PUSK_GORELKA_2:=FALSE;
	PUSK_GORELKA_3:=FALSE;
	PUSK_KASKAD_NASOSOV_1_SETEVOY:=FALSE;
	(*PUSK_KASKAD_NASOSOV_2_VNUTR:=FALSE;*)
END_IF

(*-------------------------------------------------------------------------------------ЕСЛИ АВАРИЯ НИЗКОЕ ДАВЛЕНИЕ ОТОПЛЕНИЯ*)
IF AVARIA_NIZKOE_DAVLENIE_OTOPLENIYA_SP_307 THEN
	xDO.0:=xDO0:=FALSE;(*---------------------------------------------------------------------------------------НАСОС СЕТЕВОЙ 1*)
	xDO.1:=xDO1:=FALSE;(*---------------------------------------------------------------------------------------НАСОС СЕТЕВОЙ 2*)
	xDO.2:=xDO2:=FALSE;(*----------------------------------------------------------------------НАСОС ВНУТРЕННЕГО КОНТУРА 1*)
	xDO.3:=xDO3:=FALSE;(*----------------------------------------------------------------------НАСОС ВНУТРЕННЕГО КОНТУРА 2*)

	xDO.11:=xDO11:=FALSE;(*------------------------------------------------------------------------------ГОРЕЛКА 1: ТЕРМОСТАТ*)
	xDO.12:=xDO12:=FALSE;(*------------------------------------------------------------------------------ГОРЕЛКА 2: ТЕРМОСТАТ*)
	xDO.13:=xDO13:=FALSE;(*------------------------------------------------------------------------------ГОРЕЛКА 3: ТЕРМОСТАТ*)


	PUSK_GORELKA_1:=FALSE;
	PUSK_GORELKA_2:=FALSE;
	PUSK_GORELKA_3:=FALSE;
	PUSK_KASKAD_NASOSOV_1_SETEVOY:=FALSE;
	PUSK_KASKAD_NASOSOV_2_VNUTR:=FALSE;
END_IF

(*------------------------------------------------------------------------------------------------------ЕСЛИ ВЫСОКОЕ ДАВЛЕНИЕ ГВС*)
IF AVARIA_VUSOKOE_DAVLENIE_GVS_SP_307 THEN
	xDO.4:=xDO4:=FALSE;(*---------------------------------------------------------------------------------------------НАСОС ГВС 1*)
	xDO.5:=xDO5:=FALSE;(*---------------------------------------------------------------------------------------------НАСОС ГВС 2*)

	PUSK_KASKAD_NASOSOV_3_GVS:=FALSE;
END_IF

(*--------------------------------------------------------------------------------------------------------ЕСЛИ НИЗКОЕ ДАВЛЕНИЕ ГВС*)
IF AVARIA_NIZKOE_DAVLENIE_GVS_SP_307 THEN
	xDO.4:=xDO4:=FALSE;(*---------------------------------------------------------------------------------------------НАСОС ГВС 1*)
	xDO.5:=xDO5:=FALSE;(*---------------------------------------------------------------------------------------------НАСОС ГВС 2*)

	PUSK_KASKAD_NASOSOV_3_GVS:=FALSE;
END_IF
END_ACTION
ACTION OUT_STATUS_SP_307:
(*------------------------------------------------------------------------------------------------------СТАТУС НАКОПИТЕЛЬНЫЙ БАК*)
IF EL_KL_4_NAK_BAK THEN
	STATUS_EL_KL_4_NAK_BAK_SP_307:=1;
ELSE
	STATUS_EL_KL_4_NAK_BAK_SP_307:=0;
END_IF
(*-------------------------------------------------------------------------------------СТАТУС СМЕСИТЕЛЬНЫЙ КРАН 1 ОТОПЛЕНИЕ*)
USTAVKA_ESBE_1_SP_307:=T_USTAVKA_T1;

IF ESBE_1_LESS THEN
	STATUS_ESBE_1_SP_307:=1;
END_IF
IF ESBE_1_MORE THEN
	STATUS_ESBE_1_SP_307:=2;
END_IF
IF ESBE_1_LESS=FALSE AND ESBE_1_MORE=FALSE THEN
	STATUS_ESBE_1_SP_307:=0;
END_IF
(*-----------------------------------------------------------------------------------------------СТАТУС СМЕСИТЕЛЬНЫЙ КРАН 2 ГВС*)
USTAVKA_ESBE_2_SP_307:=T_USTAVKA_T3;

IF ESBE_2_LESS THEN
	STATUS_ESBE_2_SP_307:=1;
END_IF
IF ESBE_2_MORE THEN
	STATUS_ESBE_2_SP_307:=2;
END_IF
IF ESBE_2_LESS=FALSE AND ESBE_2_MORE=FALSE THEN
	STATUS_ESBE_2_SP_307:=0;
END_IF
(*------------------------------------------------------------------------------------------------------ЭЛЕКТРОКЛАПАН 1 ПОДПИТКИ*)
IF EL_KL_1_PODPITKA_OTOPL=TRUE THEN
	STATUS_EL_KL_1_PODPITKA_SP_307:=1;
ELSE
	STATUS_EL_KL_1_PODPITKA_SP_307:=0;
END_IF
(*------------------------------------------------------------------------------------------------------ЭЛЕКТРОКЛАПАН 2 СБРОС ОТОПЛЕНИЯ*)
IF EL_KL_2_SBROS_OTOPL=TRUE THEN
	STATUS_EL_KL_2_SBROS_OTOPLENIAYA_SP_307:=1;
ELSE
	STATUS_EL_KL_2_SBROS_OTOPLENIAYA_SP_307:=0;
END_IF
(*------------------------------------------------------------------------------------------------------ЭЛЕКТРОКЛАПАН 3 СБРОС ГВС*)
IF EL_KL_3_SBROS_GVS=TRUE THEN
	STATUS_EL_KL_3_SBROS_GVS_SP_307:=1;
ELSE
	STATUS_EL_KL_3_SBROS_GVS_SP_307:=0;
END_IF
(*---------------------------------------------------------------------------------------------------------СТАТУС СЕТЕВОЙ КАСКАД 1*)
IF AVARIA_SETEVOY_NASOS_1 THEN
 	STATUS_NASOS_1_SETEVOY_1_SP_307:=2;
END_IF
IF AVARIA_SETEVOY_NASOS_2 THEN
 	STATUS_NASOS_2_SETEVOY_1_SP_307:=2;
END_IF


IF xDO.0 THEN
 	STATUS_NASOS_1_SETEVOY_1_SP_307:=1;
END_IF

IF xDO.0=FALSE AND AVARIA_SETEVOY_NASOS_1=FALSE   THEN
	STATUS_NASOS_1_SETEVOY_1_SP_307:=0;
END_IF

IF xDO.1 THEN
 	STATUS_NASOS_2_SETEVOY_1_SP_307:=1;
END_IF

IF xDO.1=FALSE AND AVARIA_SETEVOY_NASOS_2=FALSE   THEN
	STATUS_NASOS_2_SETEVOY_1_SP_307:=0;
END_IF
(*--------------------------------------------------------------------------СТАТУС ТРУБА СЕТЕВАЯ ОТОПЛЕНИЯ ЗИМНИЙ КАСКАД *)
IF  WORK_KASKAD_1_SETEVOY=FALSE AND (AVARIA_SETEVOY_NASOS_1=FALSE OR AVARIA_SETEVOY_NASOS_2=FALSE)  THEN
STATUS_TRUBA_SETEVAYA_SP_307:=0;
END_IF

IF  AVARIA_SETEVOY_NASOS_1 AND AVARIA_SETEVOY_NASOS_2 THEN
	STATUS_TRUBA_SETEVAYA_SP_307:=0;
END_IF

IF  WORK_KASKAD_1_SETEVOY=TRUE THEN
	STATUS_TRUBA_SETEVAYA_SP_307:=1;
END_IF


(*---------------------------------------------------------------------------------------------------------------СТАТУС КАСКАД ВНУТРЕННИЙ 2*)
IF AVARIA_VNUTR_NASOS_1  THEN
 	STATUS_NASOS_1_VNUTR_2_SP_307:=2;
END_IF
IF AVARIA_VNUTR_NASOS_2 THEN
 	STATUS_NASOS_2_VNUTR_2_SP_307:=2;
END_IF


IF xDO.2 THEN
 	STATUS_NASOS_1_VNUTR_2_SP_307:=1;
END_IF

IF xDO.2=FALSE AND AVARIA_VNUTR_NASOS_1=FALSE   THEN
	STATUS_NASOS_1_VNUTR_2_SP_307:=0;
END_IF

IF xDO.3 THEN
 	STATUS_NASOS_2_VNUTR_2_SP_307:=1;
END_IF

IF xDO.3=FALSE AND AVARIA_VNUTR_NASOS_2=FALSE   THEN
	STATUS_NASOS_2_VNUTR_2_SP_307:=0;
END_IF
(*-------------------------------------------------------------------------------------------------------------------СТАТУС ТРУБА ВНУТРЕННЯЯ *)
IF  WORK_KASKAD_2_VNUTR=FALSE AND (AVARIA_VNUTR_NASOS_1= FALSE OR AVARIA_VNUTR_NASOS_2=FALSE)  THEN
STATUS_TRUBA_VNUTR_SP_307:=0;
END_IF

IF  AVARIA_VNUTR_NASOS_1 AND AVARIA_VNUTR_NASOS_2 THEN
	STATUS_TRUBA_VNUTR_SP_307:=0;
END_IF

IF WORK_KASKAD_2_VNUTR=TRUE THEN
	STATUS_TRUBA_VNUTR_SP_307:=1;
END_IF
(*---------------------------------------------------------------------------------------------------------------СТАТУС КАСКАД ГВС 3*)
IF AVARIA_GVS_NASOS_1  THEN
 	STATUS_NASOS_1_GVS_3_SP_307:=2;
END_IF
IF AVARIA_GVS_NASOS_2 THEN
 	STATUS_NASOS_2_GVS_3_SP_307:=2;
END_IF


IF xDO.4 THEN
 	STATUS_NASOS_1_GVS_3_SP_307:=1;
END_IF

IF xDO.4=FALSE AND AVARIA_GVS_NASOS_1=FALSE   THEN
	STATUS_NASOS_1_GVS_3_SP_307:=0;
END_IF

IF xDO.5 THEN
 	STATUS_NASOS_2_GVS_3_SP_307:=1;
END_IF

IF xDO.5=FALSE AND AVARIA_GVS_NASOS_2=FALSE   THEN
	STATUS_NASOS_2_GVS_3_SP_307:=0;
END_IF
(*-------------------------------------------------------------------------------------------------------------------СТАТУС ТРУБА ГВС *)
IF  WORK_KASKAD_3_GVS=FALSE AND (AVARIA_GVS_NASOS_1=FALSE OR AVARIA_GVS_NASOS_2=FALSE)  THEN
STATUS_TRUBA_GVS_SP_307:=0;
END_IF

IF  AVARIA_GVS_NASOS_1 AND AVARIA_GVS_NASOS_2 THEN
	STATUS_TRUBA_GVS_SP_307:=0;
END_IF

IF WORK_KASKAD_3_GVS=TRUE THEN
	STATUS_TRUBA_GVS_SP_307:=1;
END_IF

(*--------------------------------------------------------------------------------------------СТАТУС КАСКАД КОНТУРА ПОДПИТКИ 4*)
IF AVARIA_PODPITOCHNYU_NASOS_1 THEN
 	STATUS_NASOS_1_PODPIT_4_SP_307:=2;
END_IF
IF AVARIA_PODPITOCHNYU_NASOS_2 THEN
 	STATUS_NASOS_2_PODPIT_4_SP_307:=2;
END_IF

IF xDO.6   THEN
 	STATUS_NASOS_1_PODPIT_4_SP_307:=1;
END_IF

IF xDO.6=FALSE AND AVARIA_PODPITOCHNYU_NASOS_1=FALSE   THEN
	STATUS_NASOS_1_PODPIT_4_SP_307:=0;
END_IF

IF xDO.7  THEN
 	STATUS_NASOS_2_PODPIT_4_SP_307:=1;
END_IF

IF xDO.7=FALSE AND AVARIA_PODPITOCHNYU_NASOS_2=FALSE  THEN
	STATUS_NASOS_2_PODPIT_4_SP_307:=0;
END_IF

IF AVARIA_PODPITOCHNYU_NASOS_1 AND AVARIA_PODPITOCHNYU_NASOS_2  THEN
	STATUS_TRUBA_PODPITKA_SP_307:=0;
END_IF

(*------------------------------------------------------------------------------------------------------СТАТУС ПОДПИТОЧНАЯ ТРУБА*)
IF WORK_KASKAD_4_PODPITKA
						AND (AVARIA_PODPITOCHNYU_NASOS_1=FALSE OR AVARIA_PODPITOCHNYU_NASOS_2=FALSE)  THEN
	STATUS_TRUBA_PODPITKA_SP_307:=1;
END_IF
IF WORK_KASKAD_4_PODPITKA=FALSE
						AND (AVARIA_PODPITOCHNYU_NASOS_1=FALSE OR AVARIA_PODPITOCHNYU_NASOS_2=FALSE)  THEN
	STATUS_TRUBA_PODPITKA_SP_307:=0;
END_IF

IF WORK_KASKAD_4_PODPITKA=TRUE THEN
	STATUS_TRUBA_PODPITKA_SP_307:=1;
END_IF
(*-----------------------------------------------------------------------------------------------СТАТУС ЦИРКУЛЯЦИОННЫЙ НАСОС 1*)
IF xDO.8=TRUE THEN
	STATUS_NASOS_1_CIRCULAYCIONNUY_SP_307:=1;
ELSE
	STATUS_NASOS_1_CIRCULAYCIONNUY_SP_307:=0;
END_IF
(*-----------------------------------------------------------------------------------------------СТАТУС ЦИРКУЛЯЦИОННЫЙ НАСОС 2*)
IF xDO.9=TRUE THEN
	STATUS_NASOS_2_CIRCULAYCIONNUY_SP_307:=1;
ELSE
	STATUS_NASOS_2_CIRCULAYCIONNUY_SP_307:=0;
END_IF

(*-----------------------------------------------------------------------------------------------СТАТУС ЦИРКУЛЯЦИОННЫЙ НАСОС 3*)
IF xDO.10=TRUE THEN
	STATUS_NASOS_3_CIRCULAYCIONNUY_SP_307:=1;
ELSE
	STATUS_NASOS_3_CIRCULAYCIONNUY_SP_307:=0;
END_IF
(*-------------------------------------------------------------------------------------------------------------------СТАТУС ГОРЕЛКА 1*)
IF  PUSK_GORELKA_1 AND xDO.11=TRUE THEN
	STATUS_GORELKA1_SP_307:=1;
ELSE
	STATUS_GORELKA1_SP_307:=0;
END_IF
IF AVARIA_GORELKA_1 OR S3_GORELKA_1 THEN
	STATUS_GORELKA1_SP_307:=2;
END_IF
(*-----------------------------------------------------------------------------------------------------------СТАТУС ПЛАМЯ ГОРЕЛКА 1*)
IF xDO.11=FALSE AND PUSK_GORELKA_1=FALSE  THEN
STATUS_GORENIE_1_B_M_SP_307:=0;
END_IF
IF xDO.11=TRUE AND PUSK_GORELKA_1=TRUE  THEN
STATUS_GORENIE_1_B_M_SP_307:=2;
END_IF

(*-------------------------------------------------------------------------------------------------------------------СТАТУС ГОРЕЛКА 2*)
IF  PUSK_GORELKA_2 AND xDO.12=TRUE THEN
	STATUS_GORELKA2_SP_307:=1;
ELSE
	STATUS_GORELKA2_SP_307:=0;
END_IF
IF AVARIA_GORELKA_2 OR S3_GORELKA_2 THEN
	STATUS_GORELKA2_SP_307:=2;
END_IF
(*-----------------------------------------------------------------------------------------------------------СТАТУС ПЛАМЯ ГОРЕЛКА 2*)
IF xDO.12=FALSE AND PUSK_GORELKA_2=FALSE  THEN
STATUS_GORENIE_2_B_M_SP_307:=0;
END_IF
IF xDO.12=TRUE AND PUSK_GORELKA_2=TRUE  THEN
STATUS_GORENIE_2_B_M_SP_307:=2;
END_IF

(*-------------------------------------------------------------------------------------------------------------------СТАТУС ГОРЕЛКА 3*)
IF  PUSK_GORELKA_3 AND xDO.13=TRUE THEN
	STATUS_GORELKA3_SP_307:=1;
ELSE
	STATUS_GORELKA3_SP_307:=0;
END_IF
IF AVARIA_GORELKA_3 OR S3_GORELKA_3 THEN
	STATUS_GORELKA3_SP_307:=2;
END_IF
(*-----------------------------------------------------------------------------------------------------------СТАТУС ПЛАМЯ ГОРЕЛКА 3*)
IF xDO.13=FALSE AND PUSK_GORELKA_3=FALSE  THEN
STATUS_GORENIE_3_B_M_SP_307:=0;
END_IF
IF xDO.13=TRUE AND PUSK_GORELKA_3=TRUE  THEN
STATUS_GORENIE_3_B_M_SP_307:=2;
END_IF
END_ACTION
ACTION PEREKLUCHENIE_ZIMNIY_LETNIY:
I;
(*IF ZIMNIY_KASKAD_PUSK_SP_307 OR LETNIY_KASKAD_PUSK_SP_307 THEN
	IF ZIMNIY_KASKAD_PUSK_SP_307=TRUE THEN
		CASE STEP_ZIMNIY OF
		0:
			LETNIY_KASKAD_PUSK_SP_307:=FALSE;
			STEP_ZIMNIY:=1;
			STEP_LETNIY:=0;
			(*PUSK_KASKAD_NASOSOV_1_SETEVOY:=TRUE;
			PUSK_KASKAD_NASOSOV_2_LETNIY:=FALSE;*)
		END_CASE
	END_IF
	IF LETNIY_KASKAD_PUSK_SP_307=TRUE THEN
		CASE STEP_LETNIY OF
		0:
			ZIMNIY_KASKAD_PUSK_SP_307:=FALSE;
			STEP_LETNIY:=1;
			STEP_ZIMNIY:=0;
			(*PUSK_KASKAD_NASOSOV_1_SETEVOY:=FALSE;
			PUSK_KASKAD_NASOSOV_2_LETNIY:=TRUE;*)
		END_CASE
	END_IF
END_IF

IF ZIMNIY_KASKAD_PUSK_SP_307=FALSE AND LETNIY_KASKAD_PUSK_SP_307=FALSE THEN
	STEP_LETNIY:=0;
	STEP_ZIMNIY:=0;
	(*PUSK_KASKAD_NASOSOV_1_SETEVOY:=FALSE;
	PUSK_KASKAD_NASOSOV_2_LETNIY:=FALSE;*)
END_IF
*)
END_ACTION
ACTION SBROS_ERROR:
(*------------------------------------------------------------------------------------------------СБРОС ОШИБКИ СЕТЕВОЙ КАСКАД 1*)
IF  SBROS_AVARIA_SETEVOY_KASKAD_1_SP_307=TRUE  THEN
	STEP_MAIN:=0;
	SBROS_AVARIA_SETEVOY_KASKAD_1_SP_307:=FALSE;
END_IF
(*--------------------------------------------------------------------------------------------СБРОС ОШИБКИ ВНУТРЕННИЙ КАСКАД 2*)

IF  SBROS_AVARIA_VNUTR_KASKAD_2_SP_307=TRUE  THEN
	SBROS_AVARIA_VNUTR_KASKAD_2_SP_307:=FALSE;
END_IF

(*------------------------------------------------------------------------------------------------------СБРОС ОШИБКИ КАСКАД ГВС 3*)
IF  SBROS_AVARIA_GVS_KASKAD_3_SP_307=TRUE  THEN
	SBROS_AVARIA_GVS_KASKAD_3_SP_307:=FALSE;
END_IF
(*----------------------------------------------------------------------------------------------------------СБРОС ОШИБКИ ГОРЕЛКА 1*)
IF  SBROS_AVARIA_GORELKA_1_SP_307=TRUE  THEN
	AVARIA_GORELKA_1:=FALSE;
	(*STEP_KASKAD_GORELKI:=0;
	STEP_PODOGREV_2_GORELKOY:=0;*)
	SBROS_AVARIA_GORELKA_1_SP_307:=FALSE;
END_IF
(*----------------------------------------------------------------------------------------------------------СБРОС ОШИБКИ ГОРЕЛКА 2*)
IF  SBROS_AVARIA_GORELKA_2_SP_307=TRUE  THEN
	AVARIA_GORELKA_2:=FALSE;
	(*STEP_KASKAD_GORELKI:=0;
	STEP_PODOGREV_2_GORELKOY:=0;*)
	SBROS_AVARIA_GORELKA_2_SP_307:=FALSE;
END_IF
(*----------------------------------------------------------------------------------------------------------СБРОС ОШИБКИ ГОРЕЛКА 3*)
IF  SBROS_AVARIA_GORELKA_3_SP_307=TRUE  THEN
	AVARIA_GORELKA_3:=FALSE;
	(*STEP_KASKAD_GORELKI:=0;
	STEP_PODOGREV_2_GORELKOY:=0;*)
	SBROS_AVARIA_GORELKA_3_SP_307:=FALSE;
END_IF
(*------------------------------------------------------------------------------------------СБРОС ВЫСОКОЙ ТЕМПЕРАТУРЫ КОТЕЛ 1*)
IF SBROS_AVARIA_VUSOKAYA_TEMPERATURA_KOTEL_1_SP_307 THEN
	AVARIA_VUSOKAYA_TEMPERATURA_KOTEL_1_SP_307:=FALSE;
	STEP_MAIN:=0;
	(*
	STEP_KASKAD_GORELKI:=0;
	STEP_PODOGREV_2_GORELKOY:=0;*)
END_IF
(*------------------------------------------------------------------------------------------СБРОС ВЫСОКОЙ ТЕМПЕРАТУРЫ КОТЕЛ 2*)
IF SBROS_AVARIA_VUSOKAYA_TEMPERATURA_KOTEL_2_SP_307 THEN
	AVARIA_VUSOKAYA_TEMPERATURA_KOTEL_2_SP_307:=FALSE;
	STEP_MAIN:=0;
	(*
	STEP_KASKAD_GORELKI:=0;
	STEP_PODOGREV_2_GORELKOY:=0;
	*)
END_IF
(*------------------------------------------------------------------------------------------СБРОС ВЫСОКОЙ ТЕМПЕРАТУРЫ КОТЕЛ 3*)
IF SBROS_AVARIA_VUSOKAYA_TEMPERATURA_KOTEL_3_SP_307 THEN
	AVARIA_VUSOKAYA_TEMPERATURA_KOTEL_3_SP_307:=FALSE;
	STEP_MAIN:=0;
	(*
	STEP_KASKAD_GORELKI:=0;
	STEP_PODOGREV_2_GORELKOY:=0;
	*)
END_IF
(*-------------------------------------------------------СБРОС ОШИБКИ ОБРЫВ ДАТЧИКА ТЕМПЕРАТУРЫ Т1 ПРЯМАЯ ОТОПЛЕНИЯ*)
IF  SBROS_AVARIA_OBRUV_DATCHIKA_T1_SP_307=TRUE  THEN
	AVARIA_OBRUV_DATCHIKA_T1_SP_307:=FALSE;
	SBROS_AVARIA_OBRUV_DATCHIKA_T1_SP_307:=FALSE;
END_IF
(*-----------------------------------------------------СБРОС ОШИБКИ ОБРЫВ ДАТЧИКА ТЕМПЕРАТУРЫ Т2 ОБРАТКА ОТОПЛЕНИЯ*)
IF  SBROS_AVARIA_OBRUV_DATCHIKA_T2_SP_307=TRUE  THEN
	AVARIA_OBRUV_DATCHIKA_T2_SP_307:=FALSE;
	SBROS_AVARIA_OBRUV_DATCHIKA_T2_SP_307:=FALSE;
END_IF
(*----------------------------------------------------------------СБРОС ОШИБКИ ОБРЫВ ДАТЧИКА ТЕМПЕРАТУРЫ Т3 ПРЯМАЯ ГВС*)
IF  SBROS_AVARIA_OBRUV_DATCHIKA_T3_SP_307=TRUE  THEN
	AVARIA_OBRUV_DATCHIKA_T3_SP_307:=FALSE;
	SBROS_AVARIA_OBRUV_DATCHIKA_T3_SP_307:=FALSE;
END_IF
(*---------------------------------------------------------------СБРОС ОШИБКИ ОБРЫВ ДАТЧИКА ТЕМПЕРАТУРЫ Т4 ОБРАТКА ГВС*)
IF  SBROS_AVARIA_OBRUV_DATCHIKA_T4_SP_307=TRUE  THEN
	AVARIA_OBRUV_DATCHIKA_T4_SP_307:=FALSE;
	SBROS_AVARIA_OBRUV_DATCHIKA_T4_SP_307:=FALSE;
END_IF
(*------------------------------------------------------------------СБРОС ОШИБКИ ОБРЫВ ДАТЧИКА ТЕМПЕРАТУРЫ Т5 ГОРЕЛКА 1*)
IF  SBROS_AVARIA_OBRUV_DATCHIKA_T5_SP_307=TRUE  THEN
	(*AVARIA_GORELKA_1:=FALSE;*)
	AVARIA_OBRUV_DATCHIKA_T5_SP_307:=FALSE;
	STEP_KASKAD_GORELKI:=0;
	STEP_PODOGREV_2_GORELKOY:=0;
	SBROS_AVARIA_OBRUV_DATCHIKA_T5_SP_307:=FALSE;
END_IF
(*------------------------------------------------------------------СБРОС ОШИБКИ ОБРЫВ ДАТЧИКА ТЕМПЕРАТУРЫ Т6  ГОРЕЛКА 2*)
IF  SBROS_AVARIA_OBRUV_DATCHIKA_T6_SP_307=TRUE  THEN
	(*AVARIA_GORELKA_2:=FALSE;*)
	AVARIA_OBRUV_DATCHIKA_T6_SP_307:=FALSE;
	STEP_KASKAD_GORELKI:=0;
	STEP_PODOGREV_2_GORELKOY:=0;
	SBROS_AVARIA_OBRUV_DATCHIKA_T6_SP_307:=FALSE;
END_IF
(*------------------------------------------------------------------СБРОС ОШИБКИ ОБРЫВ ДАТЧИКА ТЕМПЕРАТУРЫ Т7  ГОРЕЛКА 3*)
IF  SBROS_AVARIA_OBRUV_DATCHIKA_T7_SP_307=TRUE  THEN
	(*AVARIA_GORELKA_2:=FALSE;*)
	AVARIA_OBRUV_DATCHIKA_T7_SP_307:=FALSE;
	STEP_KASKAD_GORELKI:=0;
	STEP_PODOGREV_2_GORELKOY:=0;
	SBROS_AVARIA_OBRUV_DATCHIKA_T7_SP_307:=FALSE;
END_IF
(*-----------------------------------------------------------------------СБРОС ОШИБКИ ОБРЫВ ДАТЧИКА ТЕМПЕРАТУРЫ Т7 УЛИЦА*)
IF  SBROS_AVARIA_OBRUV_DATCHIKA_T8_SP_307=TRUE  THEN
	AVARIA_OBRUV_DATCHIKA_T8_SP_307:=FALSE;
	SBROS_AVARIA_OBRUV_DATCHIKA_T8_SP_307:=FALSE;
END_IF
(*-----------------------------------------------------------СБРОС ОШИБКИ ОБРЫВ ДАТЧИКА ДАВЛЕНИЯ Р1 ПРЯМОЙ ОТОПЛЕНИЯ*)
IF  SBROS_AVARIA_OBRUV_DATCHIKA_P1_SP_307=TRUE  THEN
	AVARIA_OBRUV_DATCHIKA_P1_SP_307:=FALSE;
	SBROS_AVARIA_OBRUV_DATCHIKA_P1_SP_307:=FALSE;
END_IF
(*----------------------------------------------------------СБРОС ОШИБКИ ОБРЫВ ДАТЧИКА ДАВЛЕНИЯ Р2 ОБРАТКИ ОТОПЛЕНИЯ*)
IF  SBROS_AVARIA_OBRUV_DATCHIKA_P2_SP_307=TRUE  THEN
	AVARIA_OBRUV_DATCHIKA_P2_SP_307:=FALSE;
	SBROS_AVARIA_OBRUV_DATCHIKA_P2_SP_307:=FALSE;
END_IF
(*---------------------------------------------------------------------СБРОС ОШИБКИ ОБРЫВ ДАТЧИКА ДАВЛЕНИЯ Р3 ПРЯМОЙ ГВС*)
IF  SBROS_AVARIA_OBRUV_DATCHIKA_P3_SP_307=TRUE  THEN
	AVARIA_OBRUV_DATCHIKA_P3_SP_307:=FALSE;
	SBROS_AVARIA_OBRUV_DATCHIKA_P3_SP_307:=FALSE;
END_IF
(*--------------------------------------------------------------------СБРОС ОШИБКИ ОБРЫВ ДАТЧИКА ДАВЛЕНИЯ Р4 ОБРАТКИ ГВС*)
IF  SBROS_AVARIA_OBRUV_DATCHIKA_P4_SP_307=TRUE  THEN
	AVARIA_OBRUV_DATCHIKA_P4_SP_307:=FALSE;
	SBROS_AVARIA_OBRUV_DATCHIKA_P4_SP_307:=FALSE;
END_IF
(*----------------------------------------------------------СБРОС ОШИБКИ ОБРЫВ ДАТЧИКА ДАВЛЕНИЯ P5  ВНУТРЕННЕГО КОНТУРА ПРЯМОЙ*)
IF  SBROS_AVARIA_OBRUV_DATCHIKA_P5_SP_307=TRUE  THEN
	AVARIA_OBRUV_DATCHIKA_P5_SP_307:=FALSE;
	SBROS_AVARIA_OBRUV_DATCHIKA_P5_SP_307:=FALSE;
END_IF
(*----------------------------------------------------------СБРОС ОШИБКИ ОБРЫВ ДАТЧИКА ДАВЛЕНИЯ P6 ВНУТРЕННЕГО КОНТУРА ПРЯМОЙ*)
IF  SBROS_AVARIA_OBRUV_DATCHIKA_P6_SP_307=TRUE  THEN
	AVARIA_OBRUV_DATCHIKA_P6_SP_307:=FALSE;
	SBROS_AVARIA_OBRUV_DATCHIKA_P6_SP_307:=FALSE;
END_IF
(*----------------------------------------------------------СБРОС ОШИБКИ ОБРЫВ ДАТЧИКА ДАВЛЕНИЯ P7 НАКОПИТЕЛЬНЫЙ БАК*)
IF  SBROS_AVARIA_OBRUV_DATCHIKA_P7_SP_307=TRUE  THEN
	AVARIA_OBRUV_DATCHIKA_P7_SP_307:=FALSE;
	SBROS_AVARIA_OBRUV_DATCHIKA_P7_SP_307:=FALSE;
END_IF
(*------------------------------------------------------------------------------------------СБРОС ВЫСОКОЕ ДАВЛЕНИЕ ОТОПЛЕНИЯ*)
IF SBROS_AVARIA_VUSOKOE_DAVLENIE_OTOPLENIYA_SP_307 THEN
	AVARIA_VUSOKOE_DAVLENIE_OTOPLENIYA_SP_307:=FALSE;
END_IF
(*--------------------------------------------------------------------------------------------СБРОС НИЗКОЕ ДАВЛЕНИЕ ОТОПЛЕНИЯ*)
IF SBROS_AVARIA_NIZKOE_DAVLENIE_OTOPLENIYA_SP_307 THEN
	AVARIA_NIZKOE_DAVLENIE_OTOPLENIYA_SP_307:=FALSE;
END_IF


(*----------------------------------------------------------------------------------------------------СБРОС ВЫСОКОЕ ДАВЛЕНИЕ ГВС*)
IF SBROS_AVARIA_VUSOKOE_DAVLENIE_GVS_SP_307 THEN
	AVARIA_VUSOKOE_DAVLENIE_GVS_SP_307:=FALSE;
END_IF
(*------------------------------------------------------------------------------------------------------СБРОС НИЗКОЕ ДАВЛЕНИЕ ГВС*)
IF SBROS_AVARIA_NIZKOE_DAVLENIE_GVS_SP_307 THEN
	AVARIA_NIZKOE_DAVLENIE_GVS_SP_307:=FALSE;
END_IF
(*----------------------------------------------------------------------------------------------СБРОС АВАРИЯ НАКОПИТЕЛЬНЫЙ БАК*)
IF SBROS_AVARIA_NAKOPITELNUY_BAK_SP_307 THEN
	AVARIA_NAKOPITELNUY_BAK_SP_307:=FALSE;
END_IF
(*-----------------------------------------------------------------------------------------------------------------------СБРОС МОДУЛЬ*)
IF SBROS_AVARIA_MODUL_SP_307 THEN
	AVARIA_MODUL_SP_307:=FALSE;
	ERROR_MODUL_SP_307:=FALSE;
	KOLICHESTVO_OBRUV_MODUL:=0;
	TIMER_MODUL_ERROR(IN:=FALSE,PT:=T#0s);
      	TIMER_MODUL_ERROR;
END_IF
(*-----------------------------------------------------------------------------------------------------------------------СБРОС ФАЗ*)
IF SBROS_AVARIA_PHASA_SP_307=TRUE THEN
	AVARIA_PHASA_SP_307:=FALSE;
END_IF
(*-----------------------------------------------------------------------------------------------------------------------СБРОС ПОЖАР*)
IF  SBROS_AVARIA_FIRE_SP_307 THEN
	AVARIA_FIRE_SP_307:=FALSE;
END_IF
(*-----------------------------------------------------------------------------------------------------------------------СБРОС ГАЗ*)
IF  SBROS_AVARIA_GAZ_SP_307 THEN
	AVARIA_GAZ_SP_307:=FALSE;
END_IF
END_ACTION
ACTION TEMPERATURNYU_REGIM:
Tpr:=TEMPERATURA_8_ULICA_AI;
IF Tpr<-27 THEN t_ustavka_T1:=95; END_IF
IF Tpr>=-27 AND Tpr<-26 THEN t_ustavka_T1:=93.6; END_IF
IF Tpr>=-26 AND Tpr<-25 THEN t_ustavka_T1:=92.2; END_IF
IF Tpr>=-25 AND Tpr<-24 THEN t_ustavka_T1:=90.8; END_IF
IF Tpr>=-24 AND Tpr<-23 THEN t_ustavka_T1:=89.4; END_IF
IF Tpr>=-23 AND Tpr<-22 THEN t_ustavka_T1:=88; END_IF
IF Tpr>=-22 AND Tpr<-21 THEN t_ustavka_T1:=86.6; END_IF
IF Tpr>=-21 AND Tpr<-20 THEN t_ustavka_T1:=85.1; END_IF
IF Tpr>=-20 AND Tpr<-19 THEN t_ustavka_T1:=83.7; END_IF
IF Tpr>=-19 AND Tpr<-18 THEN t_ustavka_T1:=82.2; END_IF
IF Tpr>=-18 AND Tpr<-17 THEN t_ustavka_T1:=80.8; END_IF
IF Tpr>=-17 AND Tpr<-16 THEN t_ustavka_T1:=79.4; END_IF
IF Tpr>=-16 AND Tpr<-15 THEN t_ustavka_T1:=77.9; END_IF
IF Tpr>=-15 AND Tpr<-14 THEN t_ustavka_T1:=76.4; END_IF
IF Tpr>=-14 AND Tpr<-13 THEN t_ustavka_T1:=75.3; END_IF
IF Tpr>=-13 AND Tpr<-12 THEN t_ustavka_T1:=73.5; END_IF
IF Tpr>=-12 AND Tpr<-11 THEN t_ustavka_T1:=72; END_IF
IF Tpr>=-11 AND Tpr<-10 THEN t_ustavka_T1:=70.4; END_IF
IF Tpr>=-10 AND Tpr<-9 THEN t_ustavka_T1:=69; END_IF
IF Tpr>=-9 AND Tpr<-8 THEN t_ustavka_T1:=67.5; END_IF
IF Tpr>=-8 AND Tpr<-7 THEN t_ustavka_T1:=65.9; END_IF
IF Tpr>=-7 AND Tpr<-6 THEN t_ustavka_T1:=64.4; END_IF
IF Tpr>=-6 AND Tpr<-5 THEN t_ustavka_T1:=62.8; END_IF
IF Tpr>=-5 AND Tpr<-4 THEN t_ustavka_T1:=61.3; END_IF
IF Tpr>=-4 AND Tpr<-3 THEN t_ustavka_T1:=59.7; END_IF
IF Tpr>=-3 AND Tpr<-2 THEN t_ustavka_T1:=58.2; END_IF
IF Tpr>=-2 AND Tpr<-1 THEN t_ustavka_T1:=56.6; END_IF
IF Tpr>=-1 AND Tpr<0 THEN t_ustavka_T1:=55; END_IF
IF Tpr>=0 AND Tpr<1 THEN t_ustavka_T1:=53.3; END_IF
IF Tpr>=1 AND Tpr<2 THEN t_ustavka_T1:=51.7; END_IF
IF Tpr>=2 AND Tpr<3 THEN t_ustavka_T1:=50.1; END_IF
IF Tpr>=3 AND Tpr<4 THEN t_ustavka_T1:=48.4; END_IF
IF Tpr>=4 AND Tpr<5 THEN t_ustavka_T1:=46.7; END_IF
IF Tpr>=5 AND Tpr<6 THEN t_ustavka_T1:=45; END_IF
IF Tpr>=6 AND Tpr<7 THEN t_ustavka_T1:=43.3; END_IF
IF Tpr>=7 AND Tpr<8 THEN t_ustavka_T1:=41.5; END_IF
IF Tpr>=8 AND Tpr<9 THEN t_ustavka_T1:=39.7; END_IF
IF Tpr>=9 AND Tpr<=10 THEN t_ustavka_T1:=38; END_IF
IF Tpr>10 THEN t_ustavka_T1:=36.1; END_IF
END_ACTION
ACTION TRASH:
I;
(*--НАРАБОТКА МИНУТ И ВЛЮЧЕНИЙ--------------------------ПЕРЕНЕС ЭТИ ПАРАМЕТРЫ В ПЕРЕМЕННЫЕ В КОНФИГУРАЦИЮ*)
(*-----------------------------------------------------------------------В СТАРЫХ ПРОГРАММАХ ХРАНИЛИСЬ В РЕТАЙН ПАМЯТИ*)
(*
	NARABOTKA_MINUT_KASKAD_1_NASOS_1_SETEVOY_SP_307: DWORD;(*--------НАРАБОТКА МИНУТ СЕТЕВОЙ НАСОС 1*)
	NARABOTKA_MINUT_KASKAD_1_NASOS_2_SETEVOY_SP_307: DWORD;(*--------НАРАБОТКА МИНУТ СЕТЕВОЙ НАСОС 2*)
	NARABOTKA_MINUT_KASKAD_2_LETNIY_NASOS_SP_307: DWORD;(*----------------НАРАБОТКА МИНУТ ЛЕТНИЙ НАСОС*)
	NARABOTKA_MINUT_KASKAD_3_NASOS_1_GVS_SP_307: DWORD;(*--------------------НАРАБОТКА МИНУТ НАСОС ГВС 1*)
	NARABOTKA_MINUT_KASKAD_3_NASOS_2_GVS_SP_307: DWORD;(*--------------------НАРАБОТКА МИНУТ НАСОС ГВС 2*)
	NARABOTKA_MINUT_KASKAD_4_NASOS_1_PODPITKA_SP_307: DWORD;(*-----НАРАБОТКА МИНУТ НАСОС ПОДПИТКА 1*)
	NARABOTKA_MINUT_KASKAD_4_NASOS_2_PODPITKA_SP_307: DWORD;(*-----НАРАБОТКА МИНУТ НАСОС ПОДПИТКА 2*)
	NARABOTKA_MINUT_KASKAD_5_NASOS_1_CIRKUL_SP_307: DWORD;(*--------НАРАБОТКА МИНУТ НАСОС ЦИРКУЛЯЦ. 1*)
	NARABOTKA_MINUT_KASKAD_5_NASOS_2_CIRKUL_SP_307: DWORD;(*--------НАРАБОТКА МИНУТ НАСОС ЦИРКУЛЯЦ. 2*)
	NARABOTKA_MINUT_GORELKA_1_SP_307:DWORD;(*---------------------------------------НАРАБОТКА МИНУТ ГОРЕЛКА 1*)
	NARABOTKA_MINUT_GORELKA_2_SP_307:DWORD;(*---------------------------------------НАРАБОТКА МИНУТ ГОРЕЛКА 2*)
	NARABOTKA_MINUT_GORELKA_3_SP_307:DWORD;(*---------------------------------------НАРАБОТКА МИНУТ ГОРЕЛКА 3*)

	KOLICHESTVO_VKLUCHENIY_KASKAD_1_NASOS_1_SETEVOY_SP_307: DWORD;(*КОЛ. ВКЛЮЧЕНИЙ СЕТЕВОЙ НАСОС 1*)
	KOLICHESTVO_VKLUCHENIY_KASKAD_1_NASOS_2_SETEVOY_SP_307: DWORD;(*КОЛ. ВКЛЮЧЕНИЙ СЕТЕВОЙ НАСОС 2*)
	KOLICHESTVO_VKLUCHENIY_KASKAD_2_LETNIY_NASOS_SP_307: DWORD;(*КОЛ. ВКЛЮЧЕНИЙ ЛЕТНИЙ НАСОС*)
	KOLICHESTVO_VKLUCHENIY_KASKAD_3_NASOS_1_GVS_SP_307: DWORD;(*КОЛ. ВКЛЮЧЕНИЙ НАСОС ГВС 1*)
	KOLICHESTVO_VKLUCHENIY_KASKAD_3_NASOS_2_GVS_SP_307: DWORD;(*КОЛ. ВКЛЮЧЕНИЙ НАСОС ГВС 2*)
	KOLICHESTVO_VKLUCHENIY_KASKAD_4_NASOS_1_PODPITKA_SP_307: DWORD;(*КОЛ. ВКЛЮЧЕНИЙ НАСОС ПОДПИТКА 1*)
	KOLICHESTVO_VKLUCHENIY_KASKAD_4_NASOS_2_PODPITKA_SP_307: DWORD;(*КОЛ. ВКЛЮЧЕНИЙ НАСОС ПОДПИТКА 2*)
	KOLICHESTVO_VKLUCHENIY_KASKAD_5_NASOS_1_CIRKUL_SP_307: DWORD;(*КОЛ. ВКЛЮЧЕНИЙ НАСОС ЦИРКУЛЯЦ. 1*)
	KOLICHESTVO_VKLUCHENIY_KASKAD_5_NASOS_2_CIRKUL_SP_307: DWORD;(*КОЛ. ВКЛЮЧЕНИЙ НАСОС ЦИРКУЛЯЦ. 2*)
	KOLICHESTVO_VKLUCHENIY_GORELKA_1_SP_307:DWORD;(*---------------------------------КОЛ. ВКЛЮЧЕНИЙ ГОРЕЛКА 1*)
	KOLICHESTVO_VKLUCHENIY_GORELKA_2_SP_307:DWORD;(*---------------------------------КОЛ. ВКЛЮЧЕНИЙ ГОРЕЛКА 2*)
	KOLICHESTVO_VKLUCHENIY_GORELKA_3_SP_307:DWORD;(*---------------------------------КОЛ. ВКЛЮЧЕНИЙ ГОРЕЛКА 3*)
*)
END_ACTION
ACTION UPRAVLENIE_GORELKOY_1:
(*------------------------------------------------------------------------------------------------------------------------------ГОРЕЛКА 1*)

(*-----------------------------------------------------------------------------------------------------------------ОСНОВНАЯ ГОРЕЛКА 1*)
IF OSNOVNAYA_GORELKA=1 THEN
	IF AVARIA_GORELKA_1=FALSE THEN
		AVARIA_OSNOVNAYA_GORELKA:=FALSE;
	END_IF
	IF AVARIA_GORELKA_1=FALSE AND AVARIA_OSNOVNAYA_GORELKA=FALSE THEN
		PUSK_GORELKA_1:=TRUE;
	ELSE
		PUSK_GORELKA_1:=FALSE;
		AVARIA_OSNOVNAYA_GORELKA:=TRUE;
	END_IF
END_IF
(*--------------------------------------------------------------------------------------------------------------------ВТОРАЯ ГОРЕЛКА 1*)
IF SECOND_GORELKA=1 THEN
	IF AVARIA_GORELKA_1=FALSE THEN
		AVARIA_SECOND_GORELKA:=FALSE;
	END_IF
	IF AVARIA_OSNOVNAYA_GORELKA=TRUE AND AVARIA_GORELKA_1=FALSE AND AVARIA_SECOND_GORELKA=FALSE THEN
		PUSK_GORELKA_1:=TRUE;
	ELSE
		PUSK_GORELKA_1:=FALSE;
	END_IF
(*-----------------------------------------------------------------------------------------------------ПОДОГРЕВ ВТОРОЙ ГОРЕЛКОЙ 1*)
	IF AVARIA_OSNOVNAYA_GORELKA=FALSE AND AVARIA_GORELKA_1=FALSE AND AVARIA_SECOND_GORELKA=FALSE THEN
		IF DELTA_TEMPERATURA_USTAVKA > PODOGREV_2_GORELKOY AND STEP_PODOGREV_SECOND_GORELKA=0 THEN
			STEP_PODOGREV_SECOND_GORELKA:=1;
		END_IF
		CASE STEP_PODOGREV_SECOND_GORELKA OF
			1:
				PUSK_GORELKA_1:=TRUE;
				IF (PODOGREV_2_GORELKOY-DELTA_TEMPERATURA_USTAVKA) >= PODOGREV_2_GORELKOY+GISTEREZIS_PODOGREV THEN
					STEP_PODOGREV_SECOND_GORELKA:=2;
				END_IF
			2:
				PUSK_GORELKA_1:=FALSE;
				STEP_PODOGREV_SECOND_GORELKA:=0;
		END_CASE
	END_IF
	IF AVARIA_GORELKA_1 THEN
		AVARIA_SECOND_GORELKA:=TRUE;
	END_IF
END_IF
(*---------------------------------------------------------------------------------------------------------------РЕЗЕРВНАЯ ГОРЕЛКА 1*)
IF RESERV_GORELKA=1 THEN
	IF AVARIA_GORELKA_1=FALSE THEN
		AVARIA_RESERV_GORELKA:=FALSE;
	END_IF
	IF AVARIA_SECOND_GORELKA=TRUE AND AVARIA_GORELKA_1=FALSE AND AVARIA_RESERV_GORELKA=FALSE THEN
		PUSK_GORELKA_1:=TRUE;
	ELSE
		PUSK_GORELKA_1:=FALSE;
	END_IF
(*-------------------------------------------------------------------------------------------------ПОДОГРЕВ РЕЗЕРВНОЙ ГОРЕЛКОЙ 1*)
	IF AVARIA_OSNOVNAYA_GORELKA=FALSE AND AVARIA_SECOND_GORELKA=FALSE AND  AVARIA_GORELKA_1=FALSE AND AVARIA_RESERV_GORELKA=FALSE THEN
		IF DELTA_TEMPERATURA_USTAVKA > PODOGREV_3_GORELKOY AND STEP_PODOGREV_RESERV_GORELKA=0 THEN
			STEP_PODOGREV_RESERV_GORELKA:=1;
		END_IF
		CASE STEP_PODOGREV_RESERV_GORELKA OF
			1:
				PUSK_GORELKA_1:=TRUE;
				IF (PODOGREV_3_GORELKOY-DELTA_TEMPERATURA_USTAVKA) >= PODOGREV_3_GORELKOY+GISTEREZIS_PODOGREV THEN
					STEP_PODOGREV_RESERV_GORELKA:=2;
				END_IF
			2:
				PUSK_GORELKA_1:=FALSE;
				STEP_PODOGREV_RESERV_GORELKA:=0;
		END_CASE
	END_IF
(*--------------------------------------------------------------ПОДОГРЕВ ВТОРОЙ ГОРЕЛКОЙ 1 ЕСЛИ ОСНОВНАЯ ВЫШЛА ИЗ СТРОЯ*)
IF (AVARIA_OSNOVNAYA_GORELKA=TRUE OR AVARIA_SECOND_GORELKA=TRUE) AND DELTA_TEMPERATURA_USTAVKA > PODOGREV_2_GORELKOY AND STEP_AVARIA_PODOGREV_RESERV_GORELKA=0 THEN
			STEP_AVARIA_PODOGREV_RESERV_GORELKA:=1;
		END_IF
		CASE STEP_AVARIA_PODOGREV_RESERV_GORELKA OF
			1:
				PUSK_GORELKA_1:=TRUE;
				IF (PODOGREV_2_GORELKOY-DELTA_TEMPERATURA_USTAVKA) >= PODOGREV_2_GORELKOY+GISTEREZIS_PODOGREV THEN
					STEP_AVARIA_PODOGREV_RESERV_GORELKA:=2;
				END_IF
			2:
				PUSK_GORELKA_1:=FALSE;
				STEP_AVARIA_PODOGREV_RESERV_GORELKA:=0;
		END_CASE

	IF AVARIA_GORELKA_1 THEN
		AVARIA_RESERV_GORELKA:=TRUE;
	END_IF
END_IF
END_ACTION
ACTION UPRAVLENIE_GORELKOY_2:
(*------------------------------------------------------------------------------------------------------------------------------ГОРЕЛКА 2*)
(*-----------------------------------------------------------------------------------------------------------------ОСНОВНАЯ ГОРЕЛКА 2*)
IF OSNOVNAYA_GORELKA=2 THEN
	IF AVARIA_GORELKA_2=FALSE THEN
		AVARIA_OSNOVNAYA_GORELKA:=FALSE;
	END_IF
	IF AVARIA_GORELKA_2=FALSE AND AVARIA_OSNOVNAYA_GORELKA=FALSE THEN
		PUSK_GORELKA_2:=TRUE;
	ELSE
		PUSK_GORELKA_2:=FALSE;
		AVARIA_OSNOVNAYA_GORELKA:=TRUE;
	END_IF
END_IF
(*---------------------------------------------------------------------------------------------------------------------ВТОРАЯ ГОРЕЛКА 2*)
IF SECOND_GORELKA=2 THEN
	IF AVARIA_GORELKA_2=FALSE THEN
		AVARIA_SECOND_GORELKA:=FALSE;
	END_IF
	IF AVARIA_OSNOVNAYA_GORELKA=TRUE AND AVARIA_GORELKA_2=FALSE AND AVARIA_SECOND_GORELKA=FALSE THEN
		PUSK_GORELKA_2:=TRUE;
	ELSE
		PUSK_GORELKA_2:=FALSE;
	END_IF
(*------------------------------------------------------------------------------------------------------ПОДОГРЕВ ВТОРОЙ ГОРЕЛКОЙ 2*)
	IF AVARIA_OSNOVNAYA_GORELKA=FALSE AND AVARIA_GORELKA_2=FALSE AND AVARIA_SECOND_GORELKA=FALSE THEN
		IF DELTA_TEMPERATURA_USTAVKA > PODOGREV_2_GORELKOY AND STEP_PODOGREV_SECOND_GORELKA=0 THEN
			STEP_PODOGREV_SECOND_GORELKA:=1;
		END_IF
		CASE STEP_PODOGREV_SECOND_GORELKA OF
			1:
				PUSK_GORELKA_2:=TRUE;
				IF (PODOGREV_2_GORELKOY-DELTA_TEMPERATURA_USTAVKA) >= PODOGREV_2_GORELKOY+GISTEREZIS_PODOGREV THEN
					STEP_PODOGREV_SECOND_GORELKA:=2;
				END_IF
			2:
				PUSK_GORELKA_2:=FALSE;
				STEP_PODOGREV_SECOND_GORELKA:=0;
		END_CASE

	END_IF
	IF AVARIA_GORELKA_2 THEN
		AVARIA_SECOND_GORELKA:=TRUE;
	END_IF
END_IF
(*-----------------------------------------------------------------------------------------------------------------РЕЗЕРВНАЯ ГОРЕЛКА 2*)
IF RESERV_GORELKA=2 THEN
	IF AVARIA_GORELKA_2=FALSE THEN
		AVARIA_RESERV_GORELKA:=FALSE;
	END_IF
	IF AVARIA_SECOND_GORELKA=TRUE AND AVARIA_GORELKA_2=FALSE AND AVARIA_RESERV_GORELKA=FALSE THEN
		PUSK_GORELKA_2:=TRUE;
	ELSE
		PUSK_GORELKA_2:=FALSE;
	END_IF
(*--------------------------------------------------------------------------------------------------ПОДОГРЕВ РЕЗЕРВНОЙ ГОРЕЛКОЙ 2*)
	IF AVARIA_OSNOVNAYA_GORELKA=FALSE AND AVARIA_SECOND_GORELKA=FALSE AND  AVARIA_GORELKA_2=FALSE AND AVARIA_RESERV_GORELKA=FALSE THEN
		IF DELTA_TEMPERATURA_USTAVKA > PODOGREV_3_GORELKOY AND STEP_PODOGREV_RESERV_GORELKA=0 THEN
			STEP_PODOGREV_RESERV_GORELKA:=1;
		END_IF
		CASE STEP_PODOGREV_RESERV_GORELKA OF
			1:
				PUSK_GORELKA_2:=TRUE;
				IF (PODOGREV_3_GORELKOY-DELTA_TEMPERATURA_USTAVKA) >= PODOGREV_3_GORELKOY+GISTEREZIS_PODOGREV THEN
					STEP_PODOGREV_RESERV_GORELKA:=2;
				END_IF
			2:
				PUSK_GORELKA_2:=FALSE;
				STEP_PODOGREV_RESERV_GORELKA:=0;
		END_CASE
	END_IF
(*--------------------------------------------------------------ПОДОГРЕВ ВТОРОЙ ГОРЕЛКОЙ 2 ЕСЛИ ОСНОВНАЯ ВЫШЛА ИЗ СТРОЯ*)

	IF (AVARIA_OSNOVNAYA_GORELKA=TRUE OR AVARIA_SECOND_GORELKA=TRUE) AND DELTA_TEMPERATURA_USTAVKA > PODOGREV_2_GORELKOY AND STEP_AVARIA_PODOGREV_RESERV_GORELKA=0 THEN
			STEP_AVARIA_PODOGREV_RESERV_GORELKA:=1;
	END_IF
		CASE STEP_AVARIA_PODOGREV_RESERV_GORELKA OF
			1:
				PUSK_GORELKA_2:=TRUE;
				IF (PODOGREV_2_GORELKOY-DELTA_TEMPERATURA_USTAVKA) >= PODOGREV_2_GORELKOY+GISTEREZIS_PODOGREV THEN
					STEP_AVARIA_PODOGREV_RESERV_GORELKA:=2;
				END_IF
			2:
				PUSK_GORELKA_2:=FALSE;
				STEP_AVARIA_PODOGREV_RESERV_GORELKA:=0;
		END_CASE

	IF AVARIA_GORELKA_2 THEN
		AVARIA_RESERV_GORELKA:=TRUE;
	END_IF
END_IF
END_ACTION
ACTION UPRAVLENIE_GORELKOY_3:
(*------------------------------------------------------------------------------------------------------------------------------ГОРЕЛКА 3*)
(*-----------------------------------------------------------------------------------------------------------------ОСНОВНАЯ ГОРЕЛКА 3*)
IF OSNOVNAYA_GORELKA=3 THEN
	IF AVARIA_GORELKA_3=FALSE THEN
		AVARIA_OSNOVNAYA_GORELKA:=FALSE;
	END_IF
	IF AVARIA_GORELKA_3=FALSE AND AVARIA_OSNOVNAYA_GORELKA=FALSE THEN
		PUSK_GORELKA_3:=TRUE;
	ELSE
		PUSK_GORELKA_3:=FALSE;
		AVARIA_OSNOVNAYA_GORELKA:=TRUE;
	END_IF
END_IF
(*--------------------------------------------------------------------------------------------------------------------ВТОРАЯ ГОРЕЛКА 3*)
IF SECOND_GORELKA=3 THEN
	IF AVARIA_GORELKA_3=FALSE THEN
		AVARIA_SECOND_GORELKA:=FALSE;
	END_IF
	IF AVARIA_OSNOVNAYA_GORELKA=TRUE AND AVARIA_GORELKA_3=FALSE AND AVARIA_SECOND_GORELKA=FALSE THEN
		PUSK_GORELKA_3:=TRUE;
	ELSE
		PUSK_GORELKA_3:=FALSE;
	END_IF
(*------------------------------------------------------------------------------------------------------ПОДОГРЕВ ВТОРОЙ ГОРЕЛКОЙ 3*)
	IF AVARIA_OSNOVNAYA_GORELKA=FALSE AND AVARIA_GORELKA_3=FALSE AND AVARIA_SECOND_GORELKA=FALSE THEN
		IF DELTA_TEMPERATURA_USTAVKA > PODOGREV_2_GORELKOY AND STEP_PODOGREV_SECOND_GORELKA=0 THEN
			STEP_PODOGREV_SECOND_GORELKA:=1;
		END_IF
		CASE STEP_PODOGREV_SECOND_GORELKA OF
			1:
				PUSK_GORELKA_3:=TRUE;
				IF (PODOGREV_2_GORELKOY-DELTA_TEMPERATURA_USTAVKA) >= PODOGREV_2_GORELKOY+GISTEREZIS_PODOGREV THEN
					STEP_PODOGREV_SECOND_GORELKA:=2;
				END_IF
			2:
				PUSK_GORELKA_3:=FALSE;
				STEP_PODOGREV_SECOND_GORELKA:=0;
		END_CASE
	END_IF
	IF AVARIA_GORELKA_3 THEN
		AVARIA_SECOND_GORELKA:=TRUE;
	END_IF
END_IF
(*-----------------------------------------------------------------------------------------------------------------РЕЗЕРВНАЯ ГОРЕЛКА 3*)
IF RESERV_GORELKA=3 THEN
	IF AVARIA_GORELKA_3=FALSE THEN
		AVARIA_RESERV_GORELKA:=FALSE;
	END_IF
	IF AVARIA_OSNOVNAYA_GORELKA=TRUE AND AVARIA_SECOND_GORELKA=TRUE AND AVARIA_GORELKA_3=FALSE AND AVARIA_RESERV_GORELKA=FALSE THEN
		PUSK_GORELKA_3:=TRUE;
	ELSE
		PUSK_GORELKA_3:=FALSE;
	END_IF
(*---------------------------------------------------------------------------------------------------ПОДОГРЕВ РЕЗЕРВНОЙ ГОРЕЛКОЙ 3*)
	IF AVARIA_OSNOVNAYA_GORELKA=FALSE AND AVARIA_SECOND_GORELKA=FALSE AND  AVARIA_GORELKA_3=FALSE AND AVARIA_RESERV_GORELKA=FALSE THEN
		IF DELTA_TEMPERATURA_USTAVKA > PODOGREV_3_GORELKOY AND STEP_PODOGREV_RESERV_GORELKA=0 THEN
			STEP_PODOGREV_RESERV_GORELKA:=1;
		END_IF
		CASE STEP_PODOGREV_RESERV_GORELKA OF
			1:
				PUSK_GORELKA_3:=TRUE;
				IF (PODOGREV_3_GORELKOY-DELTA_TEMPERATURA_USTAVKA) >= PODOGREV_3_GORELKOY+GISTEREZIS_PODOGREV THEN
					STEP_PODOGREV_RESERV_GORELKA:=2;
				END_IF
			2:
				PUSK_GORELKA_3:=FALSE;
				STEP_PODOGREV_RESERV_GORELKA:=0;
		END_CASE
	END_IF
(*--------------------------------------------------------------ПОДОГРЕВ ВТОРОЙ ГОРЕЛКОЙ 3 ЕСЛИ ОСНОВНАЯ ВЫШЛА ИЗ СТРОЯ*)

IF (AVARIA_OSNOVNAYA_GORELKA=TRUE OR AVARIA_SECOND_GORELKA=TRUE) AND DELTA_TEMPERATURA_USTAVKA > PODOGREV_2_GORELKOY AND STEP_AVARIA_PODOGREV_RESERV_GORELKA=0 THEN
			STEP_AVARIA_PODOGREV_RESERV_GORELKA:=1;
		END_IF
		CASE STEP_AVARIA_PODOGREV_RESERV_GORELKA OF
			1:
				PUSK_GORELKA_3:=TRUE;
				IF (PODOGREV_2_GORELKOY-DELTA_TEMPERATURA_USTAVKA) >= PODOGREV_2_GORELKOY+GISTEREZIS_PODOGREV THEN
					STEP_AVARIA_PODOGREV_RESERV_GORELKA:=2;
				END_IF
			2:
				PUSK_GORELKA_3:=FALSE;
				STEP_AVARIA_PODOGREV_RESERV_GORELKA:=0;
		END_CASE


	IF AVARIA_GORELKA_3 THEN
		AVARIA_RESERV_GORELKA:=TRUE;
	END_IF
END_IF
END_ACTION

(* POU PID_REGULATOR, CFC *)
FUNCTION_BLOCK PID_REGULATOR
VAR
	DIG_FILTR1: DIG_FLTR;
	PID_OTOP: PID;
	LIN_TRAFO_OTOP: LIN_TRAFO;
	VALVE_OTOP: VALVE_REG_NO_POS;
END_VAR
VAR_INPUT
	USTAVKA:REAL;
	KORREKTIROVKA:REAL;
	SBROS:BOOL;
	TEMPERATURA_IN:REAL;
	ESBE_VREMYA_HODA_ZADVIGKI:REAL;
	ESBE_MIN_VREMYA_HODA:REAL;
	ESBE_MIN_VREMYA_OSTANOVKI:REAL;
	ESBE_PROPORCIONAL:REAL;
	ESBE_INTEGRAL:REAL;
	ESBE_DIFFERINCAL:REAL;
END_VAR
VAR_OUTPUT
	LESS: BOOL;
	MORE: BOOL;
END_VAR
VAR (* helpers for the ST form of the networks *)
	_t6 : REAL;
END_VAR
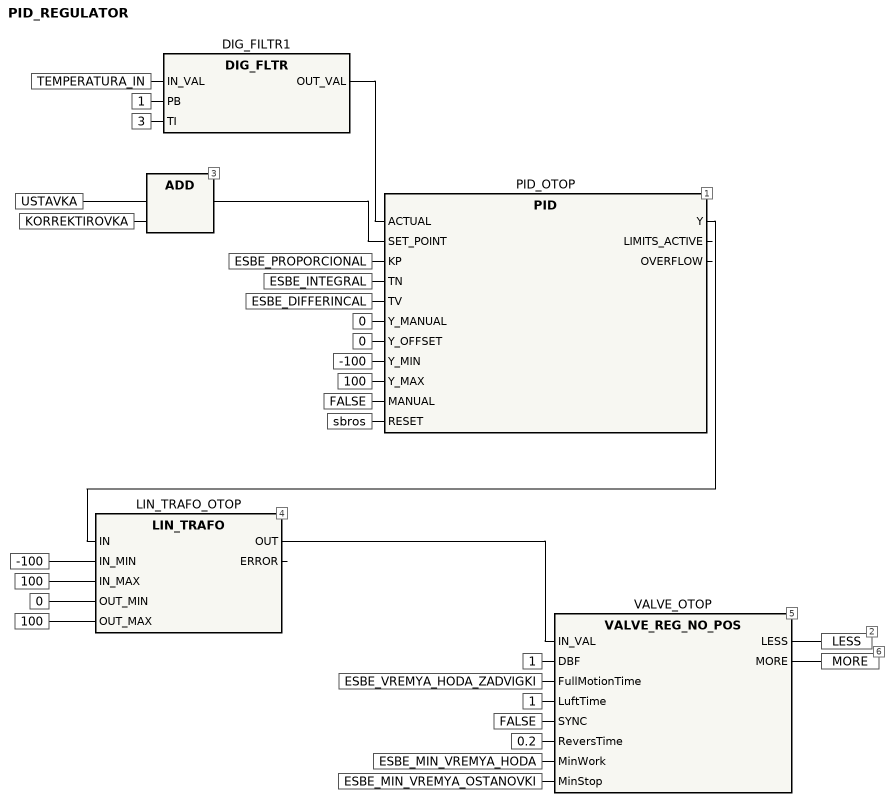
_CFC_ (* Continuous Function Chart, elements in execution order *)
#0 DIG_FILTR1:DIG_FLTR(IN_VAL: TEMPERATURA_IN, PB: 1, TI: 3)
#1 PID_OTOP:PID(ACTUAL: #0.OUT_VAL, SET_POINT: #3, KP: ESBE_PROPORCIONAL, TN: ESBE_INTEGRAL, TV: ESBE_DIFFERINCAL, Y_MANUAL: 0, Y_OFFSET: 0, Y_MIN: -100, Y_MAX: 100, MANUAL: FALSE, RESET: sbros)
#2 LESS <= #5.LESS
#3 ADD(USTAVKA, KORREKTIROVKA)
#4 LIN_TRAFO_OTOP:LIN_TRAFO(IN: #1.Y, IN_MIN: -100, IN_MAX: 100, OUT_MIN: 0, OUT_MAX: 100)
#5 VALVE_OTOP:VALVE_REG_NO_POS(IN_VAL: #4.OUT, DBF: 1, FullMotionTime: ESBE_VREMYA_HODA_ZADVIGKI, LuftTime: 1, SYNC: FALSE, ReversTime: 0.2, MinWork: ESBE_MIN_VREMYA_HODA, MinStop: ESBE_MIN_VREMYA_OSTANOVKI)
#6 MORE <= #5.MORE
_END_CFC_
(* the same logic as Structured Text *)
DIG_FILTR1(IN_VAL := TEMPERATURA_IN, PB := 1, TI := 3);
PID_OTOP(ACTUAL := DIG_FILTR1.OUT_VAL, SET_POINT := _t6, KP := ESBE_PROPORCIONAL, TN := ESBE_INTEGRAL, TV := ESBE_DIFFERINCAL, Y_MANUAL := 0, Y_OFFSET := 0, Y_MIN := -100, Y_MAX := 100, MANUAL := FALSE, RESET := sbros);
LESS := VALVE_OTOP.LESS;
_t6 := USTAVKA + KORREKTIROVKA;
LIN_TRAFO_OTOP(IN := PID_OTOP.Y, IN_MIN := -100, IN_MAX := 100, OUT_MIN := 0, OUT_MAX := 100);
VALVE_OTOP(IN_VAL := LIN_TRAFO_OTOP.OUT, DBF := 1, FullMotionTime := ESBE_VREMYA_HODA_ZADVIGKI, LuftTime := 1, SYNC := FALSE, ReversTime := 0.2, MinWork := ESBE_MIN_VREMYA_HODA, MinStop := ESBE_MIN_VREMYA_OSTANOVKI);
MORE := VALVE_OTOP.MORE;
END_FUNCTION_BLOCK

(* POU KASKAD_2_NASOSA_2_DATCHIKA_DAVLENIA, ST *)
FUNCTION_BLOCK KASKAD_2_NASOSA_2_DATCHIKA_DAVLENIA
VAR
	TP1: TP; (*-----------------------------------------------------------------------------------ПАУЗА ДЛЯ ПЕРЕПАДА ДАВЛЕНИЯ*)
	STEP:BYTE:=0; (*----------------------------------------------------------------------------------------СТАДИЯ ВЫПОЛНЕНИЯ*)
	STEP1:BYTE:=0; (*-----------------------------------------------------------------КРАТКОВРЕМЕННОЕ ПАДЕНИЕ ДАВЛЕНИЯ*)
	STEP3:BYTE:=0;(*-----------------------------------------------------------------------------------ВСПОМОГАТЕЛЬНЫЙ СТЕП*)
	STEP4:BYTE:=0;(*-----------------------------------------------------------------------------------ВСПОМОГАТЕЛЬНЫЙ СТЕП*)
	DELTA_P:REAL; (*---------------------------------------------------------------------------------РАЗНИЦА ДАВЛЕНИЙ P1 и P2*)
	STEP_OSNOVNOY: INT;(*--------------------------------------------------------------------------ВСПОМОГАТЕЛЬНЫЙ СТЕП*)
END_VAR
VAR_INPUT
	OSNOVNOY:INT;(*------------------------------------------------------------------------------------------ОСНОВНОЙ НАСОС*)
	TIME_AVARIA:TIME;(*---------------------------------------------------------------------------------------ВРЕМЯ НА АВАРИЮ*)
	P_1:REAL; (*---------------------------------------------------------------------------------------ДАВЛЕНИЕ ПОСЛЕ КАСКАДА*)
	P_2:REAL; (*--------------------------------------------------------------------------------------ДАВЛЕНИЕ ПЕРЕД КАСКАДОМ*)
	PEREPAD_DAVLENIA:REAL; (*-----------------------------------------------------------------------------ПЕРЕПАД ДАВЛЕНИЯ*)
	SBROS_ERROR: BOOL; (*----------------------------------------------------------------СБРОС ОШИБКИ КАСКАДА НАСОСОВ*)
	PUSK_NASOS:BOOL; (*------------------------------------------------------------------------------ПУСК КАСКАДА НАСОСОВ*)
END_VAR
VAR_IN_OUT
	ERROR_NASOS1: BOOL; (*----------------------------------------ОШИБКА НАСОСА 1. ХРАНИТСЯ В RETAIN КОНТРОЛЛЕРА*)
	ERROR_NASOS2: BOOL; (*----------------------------------------ОШИБКА НАСОСА 2. ХРАНИТСЯ В RETAIN КОНТРОЛЛЕРА*)
END_VAR
VAR_OUTPUT
	RELE_NASOS1:BOOL; (*--------------------------------------------------------------------------РЕЛЕ ВКЛЮЧЕНИЯ НАСОСА 1*)
	RELE_NASOS2:BOOL; (*--------------------------------------------------------------------------РЕЛЕ ВКЛЮЧЕНИЯ НАСОСА 2*)
	WORK:BOOL;(*--------------------------------------------------------------------------СТАТУС РАБОТА КАСКАДА НАСОСОВ*)
END_VAR
CASE OSNOVNOY  OF (*------------------ЗДЕСЬ ВЫБИРАЕТСЯ ОСНОВНОЙ НОСОС, И СБРАСЫВАЮТСЯ НУЖНЫЕ ПАРАМЕТРЫ*)
1:
	CASE STEP3 OF
	0:
		STEP:=0;
		STEP1:=0;
		STEP3:=1;
		STEP4:=0;
	END_CASE
2:
	CASE STEP4 OF
	0:
		STEP:=0;
		STEP1:=0;
		STEP4:=1;
		STEP3:=0;
	END_CASE;
END_CASE

IF SBROS_ERROR=TRUE  THEN(*-------------------------------------СБРОС КАСКАДА НАСОСОВ, И ОБНУЛЕНИЕ ПАРАМЕТРОВ*)
	ERROR_NASOS1:= FALSE;
	ERROR_NASOS2:=FALSE;
	STEP:=0;
	STEP1:=0;
	SBROS_ERROR:=FALSE;
END_IF

DELTA_P:=P_1-P_2;(*------------------------------------------------------------------------------РАСЧЕТ ПЕРЕПАДА ДАВЛЕНИЯ *)

IF (ERROR_NASOS1=TRUE AND ERROR_NASOS2=TRUE) THEN(*-ЕСЛИ ОШИБКА НА ДВУХ НАСОСАХ, ТО ВЫКЛЮЧИТЬ КАСКАД*)
	PUSK_NASOS:=FALSE;
END_IF


IF PUSK_NASOS=TRUE THEN(*-------------------------------------------------ЕСЛИ ДАНА КОМАНДА ПУСК КАСКАДА НАСОСОВ*)
	IF OSNOVNOY=1 THEN(*---------------------------------------------------------------------------ЕСЛИ ОСНОВНОЙ НАСОС 1*)
	IF (ERROR_NASOS1=FALSE)  OR (ERROR_NASOS2=FALSE)  THEN(*-----------ЕСЛИ НА ОДНОМ ИЗ НАСОСОВ НЕТ ОШИБКИ*)
		CASE STEP OF
			0:
				IF ERROR_NASOS1=TRUE THEN STEP:=2;(*--------------ЕСЛИ ОШИБКА 1 НАСОСА, ВКЛЮЧАЕМ СРАЗУ ВТОРОЙ*)
             			ELSE
 					RELE_NASOS1:=1;
 					RELE_NASOS2:=0;
					STEP:=1;
				END_IF
			1:
				IF DELTA_P<PEREPAD_DAVLENIA THEN	(*ЕСЛИ ПЕРЕПАД ДАВЛЕНИЯ < УСТАВКИ ТО НАЧИНАЕМ ОСЧЕТ В СЕК.*)
   				CASE STEP1 OF
					0:
						TP1(IN:=TRUE,PT:=TIME_AVARIA);
						IF  TP1.ET=TP1.PT THEN
							STEP1:=1;
							TP1(IN:=FALSE,PT:=T#0s);
      		 					TP1;
						END_IF
					1:
						IF  (ERROR_NASOS1=TRUE)  OR (DELTA_P<PEREPAD_DAVLENIA)  THEN
							RELE_NASOS1:=0;
							(*RELE_NASOS2:=1;(*--ТЕОРЕТИЧЕСКИ ЗДЕСЬ ВКЛЮЧЕНИЕ НЕ НУЖНО, ОНО БУДЕТ ВО 2 СТЕПЕ*)*)
							ERROR_NASOS1:=TRUE;
							STEP1:=0;
							STEP:=2;
						ELSE
							STEP1:=0;
						END_IF
				END_CASE
				ELSE
					TP1(IN:=FALSE,PT:=T#0s);
      		 			TP1;
				END_IF

			2:
				IF ERROR_NASOS2=TRUE THEN STEP:=4;(*-----------------ЕСЛИ ОШИБКА 2 НАСОСА, ПЕРЕХОДИМ НА 4 СТЕП*)
             			ELSE
 					RELE_NASOS1:=0;(*--------------------------------------------------------------ВЫКЛЮЧИТЬ ПЕРВЫЙ НАСОС*)
 					RELE_NASOS2:=1;(*----------------------------------------------------------------ВКЛЮЧИТЬ ВТОРОЙ НАСОС*)
					STEP:=3;
				END_IF
			3:
				IF DELTA_P<PEREPAD_DAVLENIA THEN(*--------------ЕСИЛ ДЕЛЬТА МЕНЬШЕ УСТАВКИ ПЕРЕПАДА ДАВЛЕНИЯ*)
   					CASE STEP1 OF
						0:
							TP1(IN:=TRUE,PT:=TIME_AVARIA);
							IF  TP1.ET=TP1.PT THEN
								STEP1:=1;
								TP1(IN:=FALSE,PT:=T#0s);
      		 						TP1;
							END_IF
						1:
							IF  (ERROR_NASOS2=TRUE)  OR (DELTA_P<PEREPAD_DAVLENIA)  THEN
								RELE_NASOS1:=0;
								RELE_NASOS2:=0;
								ERROR_NASOS2:=TRUE;
								STEP1:=0;
								STEP:=4;
							ELSE
								STEP1:=0;
							END_IF
					END_CASE
				ELSE
					TP1(IN:=FALSE,PT:=T#0s);
      		 			TP1;
				END_IF
			4:
				RELE_NASOS1:=0;
				RELE_NASOS2:=0;
		END_CASE
	END_IF(*-------------------------------------------------------------------------ЕСЛИ НА ОДНОМ ИЗ НАСОСОВ НЕТ ОШИБКИ*)
	END_IF(*--------------------------------------------------------------------------------------------ЕСЛИ ОСНОВНОЙ НАСОС 1*)
(*---------------------------------------------------------------------------------------------------------------------------------------*)
	IF OSNOVNOY=2 THEN(*---------------------------------------------------------------------------ЕСЛИ ОСНОВНОЙ НАСОС 2*)
	IF (ERROR_NASOS1=FALSE)  OR (ERROR_NASOS2=FALSE)  THEN(*-----------ЕСЛИ НА ОДНОМ ИЗ НАСОСОВ НЕТ ОШИБКИ*)
		CASE STEP OF
			0:
				IF ERROR_NASOS2=TRUE THEN STEP:=2;(*--------------ЕСЛИ ОШИБКА 1 НАСОСА, ВКЛЮЧАЕМ СРАЗУ ВТОРОЙ*)
             			ELSE
 					RELE_NASOS2:=1;
 					RELE_NASOS1:=0;
					STEP:=1;
				END_IF
			1:
				IF DELTA_P<PEREPAD_DAVLENIA THEN	(*ЕСЛИ ПЕРЕПАД ДАВЛЕНИЯ < УСТАВКИ ТО НАЧИНАЕМ ОСЧЕТ В СЕК.*)
   				CASE STEP1 OF
					0:
						TP1(IN:=TRUE,PT:=TIME_AVARIA);
						IF  TP1.ET=TP1.PT THEN
							STEP1:=1;
							TP1(IN:=FALSE,PT:=T#0s);
      		 					TP1;
						END_IF
					1:
						IF  (ERROR_NASOS2=TRUE)  OR (DELTA_P<PEREPAD_DAVLENIA)  THEN
							RELE_NASOS2:=0;
							(*RELE_NASOS2:=1;(*--ТЕОРЕТИЧЕСКИ ЗДЕСЬ ВКЛЮЧЕНИЕ НЕ НУЖНО, ОНО БУДЕТ ВО 2 СТЕПЕ*)*)
							ERROR_NASOS2:=TRUE;
							STEP1:=0;
							STEP:=2;
						ELSE
							STEP1:=0;
						END_IF
				END_CASE
				ELSE
					TP1(IN:=FALSE,PT:=T#0s);
      		 			TP1;
				END_IF

			2:
				IF ERROR_NASOS1=TRUE THEN STEP:=4;(*-----------------ЕСЛИ ОШИБКА 2 НАСОСА, ПЕРЕХОДИМ НА 4 СТЕП*)
             			ELSE
 					RELE_NASOS2:=0;(*--------------------------------------------------------------ВЫКЛЮЧИТЬ ПЕРВЫЙ НАСОС*)
 					RELE_NASOS1:=1;(*----------------------------------------------------------------ВКЛЮЧИТЬ ВТОРОЙ НАСОС*)
					STEP:=3;
				END_IF
			3:
				IF DELTA_P<PEREPAD_DAVLENIA THEN(*--------------ЕСИЛ ДЕЛЬТА МЕНЬШЕ УСТАВКИ ПЕРЕПАДА ДАВЛЕНИЯ*)
   					CASE STEP1 OF
						0:
							TP1(IN:=TRUE,PT:=TIME_AVARIA);
							IF  TP1.ET=TP1.PT THEN
								STEP1:=1;
								TP1(IN:=FALSE,PT:=T#0s);
      		 						TP1;
							END_IF
						1:
							IF  (ERROR_NASOS1=TRUE)  OR (DELTA_P<PEREPAD_DAVLENIA)  THEN
								RELE_NASOS2:=0;
								RELE_NASOS1:=0;
								ERROR_NASOS1:=TRUE;
								STEP1:=0;
								STEP:=4;
							ELSE
								STEP1:=0;
							END_IF
					END_CASE
				ELSE
					TP1(IN:=FALSE,PT:=T#0s);
      		 			TP1;
				END_IF
			4:
				RELE_NASOS1:=0;
				RELE_NASOS2:=0;
		END_CASE
	END_IF(*-------------------------------------------------------------------------ЕСЛИ НА ОДНОМ ИЗ НАСОСОВ НЕТ ОШИБКИ*)
	END_IF(*--------------------------------------------------------------------------------------------ЕСЛИ ОСНОВНОЙ НАСОС 2*)

ELSE(*---------------------------------------------------------------------------ЕСЛИ ДАНА КОМАНДА ПУСК КАСКАДА НАСОСОВ*)
	RELE_NASOS1:=0;
	RELE_NASOS2:=0;
	STEP:=0;
	STEP1:=0;(*-----------------------------------ДОБАВИЛ ОБНУЛЕНИЕ ВСЛЕПУЮ, НАДО ПРОВЕРИТЬ НУЖНО ЛИ ОНО ЗДЕСЬ*)
	TP1(IN:=FALSE,PT:=T#0s);
	TP1;
END_IF


(*-------------------------------------------ЕСЛИ 1 ИЛИ 2 НАСОС ВКЛЮЧЕН И ПУСК КАСКАДА ТО СТАТУС КАСКАДА "РАБОТА"*)
IF (RELE_NASOS1=1 OR RELE_NASOS2=1) AND (PUSK_NASOS=TRUE) THEN WORK:=TRUE; END_IF
(*------------------------ЕСЛИ 1 И 2 НАСОС ВЫКЛЮЧЕНЫ И ПУСК КАСКАДА ВЫКЛЮЧЕН ТО СТАТУС КАСКАДА "НЕТ РАБОТЫ"*)
IF (RELE_NASOS1=0) AND (RELE_NASOS2=0) AND (PUSK_NASOS=FALSE) THEN WORK:=FALSE; END_IF
END_FUNCTION_BLOCK

(* POU KASKAD_PODPITKA_PO_DATCHIKU_OBRATKI, ST *)
FUNCTION_BLOCK KASKAD_PODPITKA_PO_DATCHIKU_OBRATKI
VAR
	TP1: TP; (*-------------------------------------------------------------------------------------ПАУЗА ДЛЯ ПЕРЕПАДА ДАВЛЕНИЯ*)
	STEP:BYTE:=0; (*------------------------------------------------------------------------------------------СТАДИЯ ВЫПОЛНЕНИЯ*)
	STEP1:BYTE:=0; (*-------------------------------------------------------------------КРАТКОВРЕМЕННОЕ ПАДЕНИЕ ДАВЛЕНИЯ*)
	STEP3:BYTE:=0;(*-------------------------------------------------------------------------------------ВСПОМОГАТЕЛЬНЫЙ СТЕП*)
	STEP4:BYTE:=0;(*-------------------------------------------------------------------------------------ВСПОМОГАТЕЛЬНЫЙ СТЕП*)
	STEP_OSNOVNOY: INT;(*----------------------------------------------------------------------------ВСПОМОГАТЕЛЬНЫЙ СТЕП*)
END_VAR
VAR_INPUT
	OSNOVNOY:INT;(*--------------------------------------------------------------------------------------------ОСНОВНОЙ НАСОС*)
	TIME_AVARIA:TIME;(*----------------------------------------------------------------------------------------ВРЕМЯ НА АВАРИЮ*)
	P:REAL; (*------------------------------------------------------------------ДАВЛЕНИЕ ОБРАТКИ ПОДПИТЫВАЕМОГО КОНТУРА*)
	SBROS_ERROR: BOOL; (*------------------------------------------------------------------СБРОС ОШИБКИ КАСКАДА НАСОСОВ*)
	PUSK_NASOS:BOOL; (*--------------------------------------------------------------------------------ПУСК КАСКАДА НАСОСОВ*)
	USTAVKA_P:REAL;(*-----------------------------------------------------------------------------------------УСТАВКА ДАВЛЕНИЯ*)
END_VAR
VAR_IN_OUT
	ERROR_NASOS1: BOOL; (*------------------------------------------ОШИБКА НАСОСА 1. ХРАНИТСЯ В RETAIN КОНТРОЛЛЕРА*)
	ERROR_NASOS2: BOOL; (*------------------------------------------ОШИБКА НАСОСА 2. ХРАНИТСЯ В RETAIN КОНТРОЛЛЕРА*)
END_VAR
VAR_OUTPUT
	RELE_NASOS1:BOOL; (*----------------------------------------------------------------------------РЕЛЕ ВКЛЮЧЕНИЯ НАСОСА 1*)
	RELE_NASOS2:BOOL; (*----------------------------------------------------------------------------РЕЛЕ ВКЛЮЧЕНИЯ НАСОСА 2*)
	WORK:BOOL;(*----------------------------------------------------------------------------СТАТУС РАБОТА КАСКАДА НАСОСОВ*)
END_VAR
CASE OSNOVNOY  OF (*------------------ЗДЕСЬ ВЫБИРАЕТСЯ ОСНОВНОЙ НОСОС, И СБРАСЫВАЮТСЯ НУЖНЫЕ ПАРАМЕТРЫ*)
1:
	CASE STEP3 OF
	0:
		STEP:=0;
		STEP1:=0;
		STEP3:=1;
		STEP4:=0;
		TP1(IN:=FALSE,PT:=T#0s);
      	TP1;
	END_CASE
2:
	CASE STEP4 OF
	0:
		STEP:=0;
		STEP1:=0;
		STEP4:=1;
		STEP3:=0;
		TP1(IN:=FALSE,PT:=T#0s);
      	TP1;
	END_CASE;
END_CASE

IF SBROS_ERROR=TRUE  THEN(*-------------------------------------СБРОС КАСКАДА НАСОСОВ, И ОБНУЛЕНИЕ ПАРАМЕТРОВ*)
	ERROR_NASOS1:= FALSE;
	ERROR_NASOS2:=FALSE;
	STEP:=0;
	STEP1:=0;
	SBROS_ERROR:=FALSE;
END_IF


IF (ERROR_NASOS1=TRUE AND ERROR_NASOS2=TRUE) THEN(*-ЕСЛИ ОШИБКА НА ДВУХ НАСОСАХ, ТО ВЫКЛЮЧИТЬ КАСКАД*)
	PUSK_NASOS:=FALSE;
END_IF


IF PUSK_NASOS=TRUE THEN(*-------------------------------------------------ЕСЛИ ДАНА КОМАНДА ПУСК КАСКАДА НАСОСОВ*)
	IF OSNOVNOY=1 THEN(*---------------------------------------------------------------------------ЕСЛИ ОСНОВНОЙ НАСОС 1*)
	IF (ERROR_NASOS1=FALSE)  OR (ERROR_NASOS2=FALSE)  THEN(*-----------ЕСЛИ НА ОДНОМ ИЗ НАСОСОВ НЕТ ОШИБКИ*)
		CASE STEP OF
			0:
				IF ERROR_NASOS1=TRUE THEN STEP:=2;(*--------------ЕСЛИ ОШИБКА 1 НАСОСА, ВКЛЮЧАЕМ СРАЗУ ВТОРОЙ*)
             			ELSE
 					RELE_NASOS1:=1;
 					RELE_NASOS2:=0;
					STEP:=1;
				END_IF
			1:
				IF P<USTAVKA_P THEN	(*ЕСЛИ ПЕРЕПАД ДАВЛЕНИЯ < УСТАВКИ ТО НАЧИНАЕМ ОСЧЕТ В СЕК.*)
   				CASE STEP1 OF
					0:
						TP1(IN:=TRUE,PT:=TIME_AVARIA);
						IF  TP1.ET=TP1.PT THEN
							STEP1:=1;
							TP1(IN:=FALSE,PT:=T#0s);
      		 					TP1;
						END_IF
					1:
						IF  (ERROR_NASOS1=TRUE)  OR (P<USTAVKA_P)  THEN
							RELE_NASOS1:=0;
							ERROR_NASOS1:=TRUE;
							STEP1:=0;
							STEP:=2;
						ELSE
							STEP1:=0;
					END_IF
				END_CASE
				ELSE
					TP1(IN:=FALSE,PT:=T#0s);
      		 			TP1;
				END_IF

			2:
				IF ERROR_NASOS2=TRUE THEN STEP:=4;(*-----------------ЕСЛИ ОШИБКА 2 НАСОСА, ПЕРЕХОДИМ НА 4 СТЕП*)
             			ELSE
 					RELE_NASOS1:=0;(*--------------------------------------------------------------ВЫКЛЮЧИТЬ ПЕРВЫЙ НАСОС*)
 					RELE_NASOS2:=1;(*----------------------------------------------------------------ВКЛЮЧИТЬ ВТОРОЙ НАСОС*)
					STEP:=3;
				END_IF
			3:
				IF P<USTAVKA_P THEN(*--------------ЕСИЛ ДЕЛЬТА МЕНЬШЕ УСТАВКИ ПЕРЕПАДА ДАВЛЕНИЯ*)
   					CASE STEP1 OF
						0:
							TP1(IN:=TRUE,PT:=TIME_AVARIA);
							IF  TP1.ET=TP1.PT THEN
								STEP1:=1;
								TP1(IN:=FALSE,PT:=T#0s);
      		 						TP1;
							END_IF
						1:
							IF  (ERROR_NASOS2=TRUE)  OR (P<USTAVKA_P)  THEN
								RELE_NASOS1:=0;
								RELE_NASOS2:=0;
								ERROR_NASOS2:=TRUE;
								STEP1:=0;
								STEP:=4;
							ELSE
								STEP1:=0;
							END_IF
					END_CASE
				ELSE
					TP1(IN:=FALSE,PT:=T#0s);
      		 		TP1;
				END_IF
			4:
				RELE_NASOS1:=0;
				RELE_NASOS2:=0;
		END_CASE
	END_IF(*-------------------------------------------------------------------------ЕСЛИ НА ОДНОМ ИЗ НАСОСОВ НЕТ ОШИБКИ*)
	END_IF(*--------------------------------------------------------------------------------------------ЕСЛИ ОСНОВНОЙ НАСОС 1*)
(*---------------------------------------------------------------------------------------------------------------------------------------*)
	IF OSNOVNOY=2 THEN(*---------------------------------------------------------------------------ЕСЛИ ОСНОВНОЙ НАСОС 2*)
	IF (ERROR_NASOS1=FALSE)  OR (ERROR_NASOS2=FALSE)  THEN(*-----------ЕСЛИ НА ОДНОМ ИЗ НАСОСОВ НЕТ ОШИБКИ*)
		CASE STEP OF
			0:
				IF ERROR_NASOS2=TRUE THEN STEP:=2;(*--------------ЕСЛИ ОШИБКА 1 НАСОСА, ВКЛЮЧАЕМ СРАЗУ ВТОРОЙ*)
             			ELSE
 					RELE_NASOS2:=1;
 					RELE_NASOS1:=0;
					STEP:=1;
				END_IF
			1:
				IF P<USTAVKA_P THEN	(*ЕСЛИ ПЕРЕПАД ДАВЛЕНИЯ < УСТАВКИ ТО НАЧИНАЕМ ОСЧЕТ В СЕК.*)
   				CASE STEP1 OF
					0:
						TP1(IN:=TRUE,PT:=TIME_AVARIA);
						IF  TP1.ET=TP1.PT THEN
							STEP1:=1;
							TP1(IN:=FALSE,PT:=T#0s);
      		 					TP1;
						END_IF
					1:
						IF  (ERROR_NASOS2=TRUE)  OR (P<USTAVKA_P)  THEN
							RELE_NASOS2:=0;
							ERROR_NASOS2:=TRUE;
							STEP1:=0;
							STEP:=2;
						ELSE
							STEP1:=0;
						END_IF
				END_CASE
				ELSE
					TP1(IN:=FALSE,PT:=T#0s);
      		 			TP1;
				END_IF

			2:
				IF ERROR_NASOS1=TRUE THEN STEP:=4;(*-----------------ЕСЛИ ОШИБКА 2 НАСОСА, ПЕРЕХОДИМ НА 4 СТЕП*)
             	ELSE
 					RELE_NASOS2:=0;(*--------------------------------------------------------------ВЫКЛЮЧИТЬ ПЕРВЫЙ НАСОС*)
 					RELE_NASOS1:=1;(*----------------------------------------------------------------ВКЛЮЧИТЬ ВТОРОЙ НАСОС*)
					STEP:=3;
				END_IF
			3:
				IF P<USTAVKA_P THEN(*--------------ЕСИЛ ДЕЛЬТА МЕНЬШЕ УСТАВКИ ПЕРЕПАДА ДАВЛЕНИЯ*)
   					CASE STEP1 OF
						0:
							TP1(IN:=TRUE,PT:=TIME_AVARIA);
							IF  TP1.ET=TP1.PT THEN
								STEP1:=1;
								TP1(IN:=FALSE,PT:=T#0s);
      		 						TP1;
							END_IF
						1:
							IF  (ERROR_NASOS1=TRUE)  OR (P<USTAVKA_P)  THEN
								RELE_NASOS2:=0;
								RELE_NASOS1:=0;
								ERROR_NASOS1:=TRUE;
								STEP1:=0;
								STEP:=4;
							ELSE
								STEP1:=0;
							END_IF
					END_CASE
				ELSE
					TP1(IN:=FALSE,PT:=T#0s);
      		 		TP1;
				END_IF
			4:
				RELE_NASOS1:=0;
				RELE_NASOS2:=0;
		END_CASE
	END_IF(*-------------------------------------------------------------------------ЕСЛИ НА ОДНОМ ИЗ НАСОСОВ НЕТ ОШИБКИ*)
	END_IF(*--------------------------------------------------------------------------------------------ЕСЛИ ОСНОВНОЙ НАСОС 2*)





ELSE(*---------------------------------------------------------------------------ЕСЛИ ДАНА КОМАНДА ПУСК КАСКАДА НАСОСОВ*)
	RELE_NASOS1:=0;
	RELE_NASOS2:=0;
	STEP:=0;
	STEP1:=0;(*-----------------------------------ДОБАВИЛ ОБНУЛЕНИЕ ВСЛЕПУЮ, НАДО ПРОВЕРИТЬ НУЖНО ЛИ ОНО ЗДЕСЬ*)
	TP1(IN:=FALSE,PT:=T#0s);
	TP1;
END_IF


(*-------------------------------------------ЕСЛИ 1 ИЛИ 2 НАСОС ВКЛЮЧЕН И ПУСК КАСКАДА ТО СТАТУС КАСКАДА "РАБОТА"*)
IF (RELE_NASOS1=1 OR RELE_NASOS2=1) AND (PUSK_NASOS=TRUE) THEN WORK:=TRUE; END_IF
(*------------------------ЕСЛИ 1 И 2 НАСОС ВЫКЛЮЧЕНЫ И ПУСК КАСКАДА ВЫКЛЮЧЕН ТО СТАТУС КАСКАДА "НЕТ РАБОТЫ"*)
IF (RELE_NASOS1=0) AND (RELE_NASOS2=0) AND (PUSK_NASOS=FALSE) THEN WORK:=FALSE; END_IF
END_FUNCTION_BLOCK

(* POU GORELKA_ROSSEN, ST *)
FUNCTION_BLOCK GORELKA_ROSSEN
VAR_INPUT
	PUSK:BOOL;
	AVARIA:BOOL;
	RABOTA:BOOL;
	SBROS_ERROR:BOOL;
	TEMPERATURA_KOTLA:REAL;
	AVAR_TEMPERATURA:REAL;
END_VAR
VAR_IN_OUT
	ERROR_GORELKA:BOOL;
END_VAR
VAR_OUTPUT
	TERM:BOOL;
	WORK:BOOL;
END_VAR
VAR
END_VAR
IF PUSK AND AVARIA=FALSE AND ERROR_GORELKA=FALSE AND TEMPERATURA_KOTLA<AVAR_TEMPERATURA THEN
	TERM:=1;
ELSE
	TERM:=0;
END_IF

IF PUSK AND RABOTA AND ERROR_GORELKA=FALSE AND AVARIA=FALSE THEN
	WORK:=TRUE;
ELSE
	WORK:=FALSE;
END_IF



IF AVARIA=TRUE OR  TEMPERATURA_KOTLA>=AVAR_TEMPERATURA THEN
	ERROR_GORELKA:=TRUE;
	TERM:=0;
END_IF

IF SBROS_ERROR=TRUE THEN
	ERROR_GORELKA:=FALSE;
END_IF
END_FUNCTION_BLOCK

(* POU NAKOPITELNYU_BAK, ST *)
FUNCTION_BLOCK NAKOPITELNYU_BAK
VAR_INPUT
	P:REAL;(*---------------------------------------------------------------------------------------------------ДАВЛЕНИЕ С ДАТЧИКА*)
	D_MIN:REAL;(*----------------------------------------------------------------------------------------------------ДАВЛЕНИЕ В 0%*)
	D_MAX:REAL;(*-------------------------------------------------------------------------------------------------ДАВЛЕНИЕ В 100%*)
END_VAR
VAR_OUTPUT
	PROCENT_ZAPOLNENIA:INT;(*---------------------------------------------ПРОЦЕНТ ЗАПОЛНЕНИЯ НАКОПИТЕЛЬНОГО БАКА*)
END_VAR
PROCENT_ZAPOLNENIA:=REAL_TO_INT( ((P-D_MIN)*100)/(D_MAX-D_MIN));
END_FUNCTION_BLOCK

(* POU OBRYV_DATCHIKA, ST *)
FUNCTION_BLOCK OBRYV_DATCHIKA
VAR_INPUT
	VREMYA_AVARIA_OBRUV_DATCHIKA:TIME;
	ERROR:BYTE;
	SBROS_ERROR:BOOL;
END_VAR
VAR_OUTPUT
END_VAR
VAR
	STEP:INT;
	TIMER_ERROR:TP;
END_VAR
VAR_IN_OUT
	AVARIA:BOOL;
END_VAR
IF ERROR<>0 AND STEP=0 THEN
	STEP:=1;
	TIMER_ERROR(IN:=FALSE,PT:=T#0s);
      	TIMER_ERROR;
END_IF

(*-------------------------------------------------*)
IF ERROR=0 THEN
	step:=0;
END_IF
(*-------------------------------------------------*)

IF ERROR=0 AND STEP=0 THEN
	AVARIA:=FALSE;
END_IF

CASE STEP OF
1:
	TIMER_ERROR(IN:=TRUE,PT:=VREMYA_AVARIA_OBRUV_DATCHIKA);
	IF TIMER_ERROR.ET=TIMER_ERROR.PT THEN
		IF ERROR<>0 THEN
			AVARIA:=TRUE;
		END_IF
	END_IF
END_CASE;


IF  SBROS_ERROR=TRUE  THEN
	AVARIA:=FALSE;
	TIMER_ERROR(IN:=FALSE,PT:=T#0s);
      	TIMER_ERROR;
	STEP:=0;
	SBROS_ERROR:=FALSE;
END_IF
END_FUNCTION_BLOCK

(* POU MODEM, ST *)
PROGRAM MODEM
VAR
	P:POINTER TO RBDATA;
	OTVET: STRING(255);(*---------------------------------------------------------------------------------------ОТВЕТ ОТ МОДЕМА*)

	STEP_MAIN:INT;(*---------------------------------------------------------------------ГЛАВНЫЙ ЦИКЛ УПРАВЛЕНИЯ МОДЕМОМ*)
	STEP_MODEM:INT;(*---------------------------------------------------------------------ОСНОВНОЙ ЦИКЛ ОТПРАВКИ КОМАНД*)
	STEP_INTO:INT;(*--------------------------------------------------------------ВСПОМОГАТЕЛЬНЫЙ ЦИКЛ ОТПРАВКИ КОМАНД*)
	STEP_AVARIA:INT;(*---------------------------------------------ОСНОВНОЙ ЦИКЛ ОТПРАВКИ СМС СООБЩЕНИЙ ОБ АВАРИИ*)


	STR_OK:STRING;(*----------------------------------------------------------------------------------------ПОЛОЖИТЕЛЬНЙ ОТВЕТ*)
	STR_ERROR:STRING;(*----------------------------------------------------------------------------------ОТРИЦАТЕЛЬНЫЙ ОТВЕТ*)

	FIND_OK:INT;(*-------------------------------------------------------------------------------НАЙДЕН ПОЛОЖИТЕЛЬНЫЙ ОТВЕТ*)
	FIND_ERROR:INT;(*---------------------------------------------------------------------------НАЙДЕН ОТРИЦАТЕЛЬНЫЙ ОТВЕТ*)

	TIME_ZADERGKA_OTPRAVKI_SOOBSHENIY:TIME:=T#30S;(*----------------ВРЕМЯ ЗАДЕРЖКИ ПОСЛЕ ВКЛЮЧЕНИЯ МОДЕМА*)
	ZADERGKA_PEREHODA:TIME:=T#200MS;(*-------------------------------------------------------ВРЕМЯ ЗАДЕРЖКИ ПЕРЕХОДА*)
	OGIDANIE_OTVETA:TIME:=T#10S;(*----------------------------------------------------------------ВРЕМЯ ОЖИДАНИЯ ОТВЕТА*)

	TIMER_ZADERGKA_OTPRAVKI_SOOBSHENIY:TP;(*----------------------ЗАДЕРЖКА ДЛЯ ТОГО ЧТО БЫ МОДЕМ ПРОГРУЗИЛСЯ*)
	PAUSA:TP;(*------------------------------------------------------------------------ПАУЗА ДЛЯ ПЕРЕХОДА НА СЛЕДУЮЩИЙ ШАГ*)
	TIMER_OTVET:TP;(*--------------------------------------------------------------------------------ТАЙМЕР ОЖИДАНИЯ ОТВЕТА*)

	POPUTKA:INT;(*------------------------------------------------------КОЛИЧЕСТВО ПОПЫТОК ЕСЛИ ОТРИЦАТЕЛЬНЫЙ ОТВЕТ*)
	POPUTKA_PO_VREMENI:INT;(*------------------------------КОЛИЧЕСТВО ПОПЫТОК ЕСЛИ НЕ УКЛАДЫВАЕТСЯ ПО ВРЕМЕНИ*)
	POPUTKA_AVARIA: INT;(*-----------------------------КОЛИЧЕСТВО ПОПЫТОК ЕСЛИ ОТРИЦАТЕЛЬНЫЙ ОТВЕТ ПРИ АВАРИИ*)
	POPUTKA_PO_VREMENI_AVARIA: INT;(*-----КОЛИЧЕСТВО ПОПЫТОК ЕСЛИ НЕ УКЛАДЫВАЕТСЯ ПО ВРЕМЕНИ ПРИ АВАРИИ*)

	SMS_MODEM_1:INT;
	NUMBER:STRING(80);
	NUMBER1:STRING(80);(*------------------------------------------------------------------------------------------------ТЕЛЕФОН 1*)
	NUMBER2:STRING(80);(*------------------------------------------------------------------------------------------------ТЕЛЕФОН 2*)
	NUMBER3:STRING(80);(*------------------------------------------------------------------------------------------------ТЕЛЕФОН 3*)
	TEL:INT:=1;(*-------------------------------------------------------------------------------ПЕРЕМЕННАЯ ДЛЯ СМЕНЫ НОМЕРОВ*)


	TIMER_SEND_OK:TP;
	TIME_SEND_OK:TIME:=T#10M;
	FIND_TIMER_SEND_OK:INT;
	STRING_SEND_OK:STRING:='SEND OK$R$NHTTP/1.1 200 OK';
(*-----------------------------------------------------------------------------------------------------------------------------------------*)
	step_set_byte:INT;
	step_SMENA_NOMERA:INT;
	step_otvet2:INT;

	KOL_SMS:INT;
	step_number:INT;

	TIMER_DAY:TP;
	TIMER_REBOOT:TP;
	REBOOT:INT;
	I:INT;
	COMMAND:STRING;

	OTVET2: STRING(255);
	STRING_SEND:STRING(255);
	STRING_SEND_2:STRING(255);
	STRING_SEND_3:STRING(255);
	STRING_SEND_4:STRING(255);
	STRING_SEND_5:STRING(255);
	STRING_SEND_6:STRING(255);
	STRING_SEND_7:STRING(255);
	STRING_SEND_8:STRING(255);
	STRING_SEND_9:STRING(255);
	STRING_SEND_10:STRING(255);
	STRING_SEND_11:STRING(255);
	STRING_SEND_12:STRING(255);
	STRING_SEND_13:STRING(255);
	STRING_SEND_14:STRING(255);
	STRING_SEND_15:STRING(255);
	STRING_SEND_16:STRING(255);

	STR_ZAVIS:STRING:='SIM800 R13.08';
	LEN_STRING_SEND_vsego:INT;
	LEN_STRING_SEND_2:INT;
	LEN_STRING_SEND_3:INT;
	LEN_STRING_SEND_4:INT;
	LEN_STRING_SEND_5:INT;
	LEN_STRING_SEND_6:INT;
	LEN_STRING_SEND_7:INT;
	LEN_STRING_SEND_8:INT;
	LEN_STRING_SEND_9:INT;
	LEN_STRING_SEND_10:INT;
	LEN_STRING_SEND_11:INT;
	LEN_STRING_SEND_12:INT;
	LEN_STRING_SEND_13:INT;
	LEN_STRING_SEND_14:INT;
	LEN_STRING_SEND_15:INT;
	LEN_STRING_SEND_16:INT;







	ERROR:BOOL;





	STR_FIND:INT;


	(*-------------------------------------------------------------------------------------*)
	AVAR_SMS:BOOL;
	I1:INT;



	KOL_TELEFONOV:INT:=2;
	POPUTKA_POSLE_REBOOT:INT;
	(*-------------------------------------------------------------------------------------*)
	(*AVARIA_NASOS_1_KASKAD_1_SETEVOY_SP_307:BOOL;
	AVARIA_NASOS_2_KASKAD_1_SETEVOY_SP_307:BOOL;
	AVARIA_NASOS_1_KASKAD_2_VNUTR_KONTUR_SP_307:BOOL;
	AVARIA_NASOS_2_KASKAD_2_VNUTR_KONTUR_SP_307:BOOL;
	AVARIA_NASOS_1_KASKAD_3_PODPITKA_SP_307:BOOL;
	AVARIA_NASOS_2_KASKAD_3_PODPITKA_SP_307:BOOL;
	AVARIA_GORELKA_1_SP_307:BOOL;
	AVARIA_GORELKA_2_SP_307:BOOL;
	AVARIA_GORELKA_3_SP_307:BOOL;
	AVARIA_VKLUCHITE_GORELKA_1_SP_307:BOOL;
	AVARIA_VKLUCHITE_GORELKA_2_SP_307:BOOL;
	AVARIA_VKLUCHITE_GORELKA_3_SP_307:BOOL;
	AVARIA_PHASA_SP_307:BOOL;
	AVARIA_FIRE_SP_307:BOOL;
	AVARIA_GAS_SP_307:BOOL;
	AVARIA_ZAP_KRAN_1_SP_307:BOOL;
	AVARIA_ZAP_KRAN_2_SP_307:BOOL;
	AVARIA_ZAP_KRAN_3_SP_307:BOOL;
	AVARIA_VYSOKOE_DAVL_OTOP_SP_307:BOOL;
	AVARIA_NIZKOE_DAVL_OTOP_SP_307:BOOL;
	AVARIA_VYSOKOE_DAVL_VNUTR_KONTURA_SP_307:BOOL;
	AVARIA_NIZKOE_DAVL_VNUTR_KONTURA_SP_307:BOOL;
	AVARIA_VYSOKOE_DAVL_PODPITKI_SP_307:BOOL;
	AVARIA_NIZKOE_DAVL_PODPITKI_SP_307:BOOL;
	AVARIA_OBRUV_DATCHIKA_TEMP1_PR_OTOP_SP_307:BOOL;
	AVARIA_OBRUV_DATCHIKA_TEMP2_OBR_OTOP_SP_307:BOOL;
	AVARIA_OBRUV_DATCHIKA_TEMP3_OBR_VNUTR_KONTURA_SP_307:BOOL;
	AVARIA_OBRUV_DATCHIKA_TEMP4_KOTEL_1_SP_307:BOOL;
	AVARIA_OBRUV_DATCHIKA_TEMP5_KOTEL_2_SP_307:BOOL;
	AVARIA_OBRUV_DATCHIKA_TEMP6_KOTEL_3_SP_307:BOOL;
	AVARIA_OBRUV_DATCHIKA_TEMP7_ULICA_SP_307:BOOL;
	AVARIA_OBRUV_DATCHIKA_DAVL1_PR_OTOP_SP_307:BOOL;
	AVARIA_OBRUV_DATCHIKA_DAVL2_OBR_OTOP_SP_307:BOOL;
	AVARIA_OBRUV_DATCHIKA_DAVL3_PR_VNUTR_KONTUR_SP_307:BOOL;
	AVARIA_OBRUV_DATCHIKA_DAVL4_OBR_VNUTR_KONTUR_SP_307:BOOL;
	AVARIA_OBRUV_DATCHIKA_DAVL5_PR_PODPITKI_SP_307:BOOL;
	AVARIA_OBRUV_DATCHIKA_DAVL6_OBR_PODPITKI_SP_307:BOOL;
	AVARIA_OBRUV_DATCHIKA_DAVL7_NAK_BAK_SP_307:BOOL;
	AVARIA_VYSOKAYA_TEMPERATURA_KOTEL_1_SP_307:BOOL;
	AVARIA_VYSOKAYA_TEMPERATURA_KOTEL_2_SP_307:BOOL;
	AVARIA_VYSOKAYA_TEMPERATURA_KOTEL_3_SP_307:BOOL;

	DAV1_PR_OTOP_AI_SP_307:REAL:=2.42345245;
	DAV2_OBR_OTOP_AI_SP_307:REAL:=34.423452345;
	DAV3_PR_NAGREV_KONT_AI_SP_307:REAL:=222.42345245;
	DAV4_OBR_NAGREV_KONT_AI_SP_307:REAL:=1.323452;
	DAV5_PR_PODPIT_AI_SP_307:REAL:=20;
	DAV6_OBR_PODPIT_AI_SP_307:REAL:=5;
	DAV7_NAK_BAK_AI_SP_307:REAL:=88;

	TEMP1_PR_OTOP_AI_SP_307:REAL:=2.423452;
	TEMP2_OBR_OTOP_AI_SP_307:REAL:=2.4234523;
	TEMP3_OBR_NAGR_KONT_AI_SP_307:REAL:=2.434545;
	TEMP4_KOTEL_1_AI_SP_307:REAL:=2.454654;
	TEMP5_KOTEL_2_AI_SP_307:REAL:=2.456476;
	TEMP6_KOTEL_3_AI_SP_307:REAL:=2.4245;
	TEMP7_ULICA_AI_SP_307:REAL:=2.4679769;

	status_nasos1_setevoy_1_sp_307:INT;
	status_nasos2_setevoy_1_sp_307:INT;
	status_truba_setevoy_sp_307:INT;
	status_nasos1_kontur_nagrev_2_sp_307:INT;
	status_nasos2_kontur_nagrev_2_sp_307:INT;
	status_truba_kontr_nagrev_sp_307:INT;
	status_nasos1_podpit_3_sp_307:INT;
	status_nasos2_podpit_3_sp_307:INT;
	status_truba_podpit_sp_307:INT;
	status_zadvigki_1_sp307:INT;
	status_zadvigki_2_sp307:INT;
	status_zadvigki_3_sp307:INT;
	STATUS_GORELKA1_SP_307:INT;
	STATUS_GORELKA2_SP_307:INT;
	STATUS_GORELKA3_SP_307:INT;
	STATUS_GORENIE_B_M_sp_307:INT;
	STATUS_TRUBA_POSLE_KOTEL_1_SP_307:INT;
	STATUS_TRUBA_POSLE_KOTEL_2_SP_307:INT;
	STATUS_TRUBA_POSLE_KOTEL_3_SP_307:INT;
	STATUS_EL_KL_1_PODP_KONT_NAGR_SP_307:INT;
	STATUS_EL_KL_2_PODP_OTOP_SP_307:INT;
	STATUS_EL_KL_3_SBROS_VNUTR_KONTUR_SP_307:INT;
	STATUS_EL_KL_4_SBROS_OTOP_SP_307:INT;
	STATUS_EL_KL_5_NAK_BAK_SP_307:INT;
	STATUS_EL_KL_6_OTSECH_GAS_SP_307:INT;
	PROCENT_NAK_BAK:INT;
	STATUS_ESBE_SP_307:INT;
*)
	A1_R: R_TRIG;
	A2_R: R_TRIG;
	A3_R: R_TRIG;
	A4_R: R_TRIG;
	A5_R: R_TRIG;
	A6_R: R_TRIG;
	A7_R: R_TRIG;
	A8_R: R_TRIG;
	A9_R: R_TRIG;
	A10_R: R_TRIG;
	A11_R: R_TRIG;
	A12_R: R_TRIG;
	A13_R: R_TRIG;
	A14_R: R_TRIG;
	A15_R: R_TRIG;
	A16_R: R_TRIG;
	A17_R: R_TRIG;
	A18_R: R_TRIG;
	A19_R: R_TRIG;
	A20_R: R_TRIG;
	A21_R: R_TRIG;
	A22_R: R_TRIG;
	A23_R: R_TRIG;
	A24_R: R_TRIG;
	A25_R: R_TRIG;
	A26_R: R_TRIG;
	A27_R: R_TRIG;
	A28_R: R_TRIG;
	A29_R: R_TRIG;
	A30_R: R_TRIG;
	A31_R: R_TRIG;
	A32_R: R_TRIG;
	A33_R: R_TRIG;
	A34_R: R_TRIG;
	A35_R: R_TRIG;
	A36_R: R_TRIG;
	A37_R: R_TRIG;
	A38_R: R_TRIG;
	A39_R: R_TRIG;
	A40_R: R_TRIG;
	A41_R: R_TRIG;
	A42_R: R_TRIG;
	A43_R: R_TRIG;
	A44_R: R_TRIG;
	A45_R: R_TRIG;

